(* CODESYS project SPT_MotionControl.library
   Placeholder: SPT Motion Control
   Title: SPT Motion Control
   Version: 3.1.0
   Company: Beckhoff Automation LLC

Project tree, tasks and I/O mapping:
  libraries: SPT Base Types, * (Beckhoff Automation LLC); Tc2_Math, * (Beckhoff Automation GmbH); Tc2_MC2, * (Beckhoff Automation GmbH); Tc2_MC2_Camming, * (Beckhoff Automation GmbH); Tc2_MC2_Drive, * (Beckhoff Automation GmbH); Tc2_Standard, * (Beckhoff Automation GmbH); Tc2_System, * (Beckhoff Automation GmbH); Tc3_MC2_AdvancedHoming, * (Beckhoff Automation GmbH); Tc3_Module, * (Beckhoff Automation GmbH)
  DUTs/
    data type E_CamAxisState
    data type E_CamSyncMode
    data type ST_AbsHomeParameters
    data type ST_CamParameters
    data type ST_CamPoints
    data type ST_StepBlockLagBasedParameters
  Function Blocks/
    Hardware Utilities/
      function block FB_ResetRoutine_CoEDrive [ST]: Axis, CyclicLogic, Execute
      function block FB_ResetRoutine_SoEDrive [ST]: Axis, CyclicLogic, Execute
    Homing Routines/
      function block FB_HomeRoutine_AbsHoming [ST]: Axis, CyclicLogic, Execute, Parameters
      function block FB_HomeRoutine_HardStop [ST]: Axis, CyclicLogic, Execute, HomePosition, Parameters
      function block FB_HomeRoutine_SetPosition [ST]: Axis, CyclicLogic, Execute, HomePosition
      function block FB_HomeRoutine_SetZeroHere [ST]: Axis, CyclicLogic, Execute
    function block FB_BasicAxis [ST]: Disable, Enable, Home, Jog, MoveAbsolute, MoveModulo, MoveRelative, MoveVelocity, Reset, Stop, WriteBoolParameter, WriteParameter, Acceleration, Deceleration, Jerk, Velocity, ActualAcceleration, ActualPosition, ActualPositionModulo, ActualTorque, ActualVelocity, PositionLag, SetAcceleration, SetPosition, SetPositionModulo, SetVelocity, Enabled, InPosition, Stopped, Axis, HomeMethod, InhibitFeedNegative, InhibitFeedPositive, Override, ResetMethod, CyclicLogic, CallFBs, Initialize, AxisParameters
    function block FB_BasicSlaveAxis [ST]: Home, MoveAbsolute, MoveModulo, MoveRelative, MoveVelocity, Reset, GearIn, GearOut, InGear, Master1, Master2, Master3, Master4, RatioMaster1, RatioMaster2, RatioMaster3, RatioMaster4, Stop, CyclicLogic, CallFBs, Initialize
    function block FB_CamSlaveAxis [ST]: Home, MoveModulo, Reset, Stop, CamParameters, ChangeMode, FindSlavePos, FindSyncPos, InSync, Master, RunningTable, StartCouple, StartSync, SyncPos, UpdateTable, CyclicLogic, CallFBs, Initialize
    function block FB_RingBuffer_MCMoveAbsolute [ST]: CurrentFB, GetNewFB
    function block FB_RingBuffer_MCMoveModulo [ST]: CurrentFB, GetNewFB
    function block FB_RingBuffer_MCMoveRelative [ST]: CurrentFB, GetNewFB
    function block FB_RingBuffer_MCMoveVelocity [ST]: CurrentFB, GetNewFB
  Interfaces/
    interface I_BasicAxis: Disable, Enable, Home, Jog, MoveAbsolute, MoveModulo, MoveRelative, MoveVelocity, Reset, Stop, WriteBoolParameter, WriteParameter, Acceleration, Deceleration, Jerk, Velocity, ActualAcceleration, ActualPosition, ActualPositionModulo, ActualTorque, ActualVelocity, PositionLag, SetAcceleration, SetPosition, SetPositionModulo, SetVelocity, Enabled, InPosition, Stopped, Axis, HomeMethod, InhibitFeedNegative, InhibitFeedPositive, Override, ResetMethod
    interface I_BasicSlaveAxis: GearIn, GearOut, InGear, Master1, Master2, Master3, Master4, RatioMaster1, RatioMaster2, RatioMaster3, RatioMaster4
    interface I_CamSlaveAxis: CamParameters, ChangeMode, FindSlavePos, FindSyncPos, InSync, Master, RunningTable, StartCouple, StartSync, SyncPos, UpdateTable
    interface I_MotionSequence: Axis, Execute
  Project Information/
    function F_GetCompany [ST]
    function F_GetTitle [ST]
    function F_GetVersion [ST]
  Version/
    global variables Global_Version
  global variables Parameters_MotionControl
*)

// DUTs/E_CamAxisState
{attribute 'qualified_only'}
{attribute 'strict'}
TYPE E_CamAxisState : (
        eCamAxisState_Disabled := 0,
        eCamAxisState_ReadMasterParameters,
        eCamAxisState_ReadSlaveParameters,
        eCamAxisState_AxisInitDone,
        eCamAxisState_WaitForCommand,
        eCamAxisState_DecoupleBeforeStart,
        eCamAxisState_CheckTableSelect,
        eCamAxisState_LoadCamTable,
        eCamAxisState_CheckAxisStatus,
        eCamAxisState_ReadSlaveDynamics,
        eCamAxisState_DetermineSyncMove,
        eCamAxisState_SlaveSyncMove,
        eCamAxisState_CoupleSlave,
        eCamAxisState_SetChangeMode,
        eCamAxisState_WaitForChangeCommand,
        eCamAxisState_WriteNewTable,
        eCamAxisState_WaitForActive,
        //eCamAxisState_DecoupleSlave,

        //eCamAxisState_HaltSlave,
        eCamAxisState_Error
    ) UDINT;
END_TYPE

// DUTs/E_CamSyncMode
{attribute 'qualified_only'}
{attribute 'strict'}
TYPE E_CamSyncMode : (
        eCamSyncMode_ShortestWay    := 0, // Move the Shortest Distance
        eCamSyncMode_Forward        := 1, // Move Only in the Forward Direction
        eCamSyncMode_Reverse        := 2, // Move Only in the Reverse Direction
        eCamSyncMode_Window_Forward := 3, // Move Shortest Distance If In Window Else Move Forward
        eCamSyncMode_Window_Reverse := 4  // Move Shortest Distance If In Window Else Move Reverse
    );
END_TYPE

// DUTs/ST_AbsHomeParameters
TYPE ST_AbsHomeParameters :
    STRUCT
        PositionBias           : LREAL;
        PositionLimit_Positive : LREAL;
        PositionLimit_Negative : LREAL;
    END_STRUCT
END_TYPE

// DUTs/ST_CamParameters
TYPE ST_CamParameters :
    STRUCT
        // Table Must Be Constructed of Motion Functions
        MasterPos    : LREAL         := 0.1;                                    // Position of Master For Which Corresponding Slave Position Is Found For
        SyncMode     : E_CamSyncMode := E_CamSyncMode.eCamSyncMode_ShortestWay; // Specifies Which Direction Slave Moves To Synchronize With the Master
        SyncWindow   : LREAL         := 10.0;                                   // Used In Conjunction With Sync Mode
        SyncVelocity : LREAL         := 10.0;                                   // Used When Slave Moves To Synchronization Position
        SyncAccel    : LREAL         := 100.0;                                  // Used When Slave Moves To Synchronization Position
        SyncDecel    : LREAL         := 100.0;                                  // Used When Slave Moves To Synchronization Position
        SyncJerk     : LREAL         := 1000.0;                                 // Used When Slave Moves To Synchronization Position

        //EmergencyDecel : LREAL         := 1000.0;                                 // Rate At Which Slave Stops On Loss of Function Block Enable or Error

        //EmergencyJerk  : LREAL         := 10000.0;                                // Rate At Which Slave Stops On Loss of Function Block Enable or Error
        TableSelect   : UDINT     := 1; // Selects Which of Five Cam Tables To Use
        CamTableId    : MC_CAM_ID := 1; // Make Sure All Your Id's are Unique
        CamTable      : ARRAY[1..Parameters_MotionControl.CAM_SLAVE_AXIS_TABLES] OF ST_CamPoints;
        Periodic      : BOOL         := TRUE;
        MasterOffset  : LREAL        := 0.0;
        SlaveOffset   : LREAL        := 0.0;
        MasterScaling : LREAL        := 1.0;
        SlaveScaling  : LREAL        := 1.0;
        StartMode     : MC_StartMode := MC_STARTMODE_ABSOLUTE;
        BufferMode    : MC_BufferMode;
        CamInOptions  : ST_CamInOptions;
        ChangeOptions : ST_CamInOptions; // Used for MC_SetCamOnlineChangeMode; Change Mode is Set After Cam In
    END_STRUCT
END_TYPE

// DUTs/ST_CamPoints
TYPE ST_CamPoints :
    STRUCT
        Points         : ARRAY[1..Parameters_MotionControl.CAM_SLAVE_AXIS_MAX_CAM_POINTS] OF MC_MotionFunctionPoint; // Array of Points 
        NumberOfPoints : DINT;                                                                                   // Quantity of Points 
    END_STRUCT
END_TYPE

// TYPE MC_MotionFunctionType

// 	MOTIONFUNCTYPE_NOTDEF,

//	MOTIONFUNCTYPE_POLYNOM1

//	MOTIONFUNCTYPE_POLYNOM3

//	MOTIONFUNCTYPE_POLYNOM5								Rest to Rest

//	MOTIONFUNCTYPE_POLYNOM8

// 	MOTIONFUNCTYPE_SINUSLINIE

//	MOTIONFUNCTYPE_MODSINUSLINIE

//	MOTIONFUNCTYPE_BESTEHORN

//	MOTIONFUNCTYPE_BESCHLTRAPEZ

//	MOTIONFUNCTYPE_POLYNOM5_MM						Motion to Motion

//	MOTIONFUNCTYPE_SINUS_GERADE_KOMBI

// 	MOTIONFUNCTYPE_HARMONIC_KOMBI_RT

//	MOTIONFUNCTYPE_HARMONIC_KOMBI_TR

//	MOTIONFUNCTYPE_HARMONIC_KOMBI_VT

//	MOTIONFUNCTYPE_HARMONIC_KOMBI_TV

//	MOTIONFUNCTYPE_BESCHLTRAPEZ_RT

//	MOTIONFUNCTYPE_BESCHLTRAPEZ_RT

//	MOTIONFUNCTYPE_MODSINUSLINIE_VV

//	MOTIONFUNCTYPE_POLYNOM7_MM

//	MOTIONFUNCTYPE_POLYNOM6STP

//	MOTIONFUNCTYPE_POLYNOM6WDP

//	MOTIONFUNCTYPE_STEPFUNCTION

// TYPE MC_MotionFunctionPoint

//	MOTIONPOINTTYPE_IGNORE

//	MOTIONPOINTTYPE_REST				Vel = 0 and Accel = 0

//	MOTIONPOINTTYPE_VELOCITY		Vel = V and Accel = 0

//	MOTIONPOINTTYPE_TURN				Vel = 0 and Accel = A

//	MOTIONPOINTTYPE_MOTION			Vel = V and Accel = A

//	MOTIONPOINTTYPE_ADD

//	MOTIONPOINTTYPE_ACTIVATION

// DUTs/ST_StepBlockLagBasedParameters
TYPE ST_StepBlockLagBasedParameters :
    STRUCT
        Direction              : MC_Home_Direction := mcNegativeDirection;
        Velocity               : LREAL             := 10;
        Acceleration           : LREAL             := 100;
        Deceleration           : LREAL             := 100;
        Jerk                   : LREAL             := 1000;
        DetectionVelocityLimit : LREAL             := 5;
        DetectionVelocityTime  : TIME              := T#500MS;
        TimeLimit              : TIME;
        DistanceLimit          : LREAL;
        TorqueLimit            : LREAL            := 10;
        LagLimit               : LREAL            := 10;
        Options                : ST_Home_Options3 := (InstantLagReduction := TRUE);
    END_STRUCT
END_TYPE

// Version/Global_Version
{attribute 'TcGenerated'}
{attribute 'no-analysis'}
{attribute 'linkalways'}
// This function has been automatically generated from the project information.
VAR_GLOBAL CONSTANT
	{attribute 'const_non_replaced'}
	stLibVersion_SPT_Motion_Control : ST_LibVersion := (iMajor := 3, iMinor := 1, iBuild := 0, iRevision := 0, nFlags := 1, sVersion := '3.1.0');
END_VAR

// Parameters_MotionControl
{attribute 'qualified_only'}
VAR_GLOBAL CONSTANT
    ALLOW_UNLINKED_NC_AXES : BOOL := FALSE;
	    CAM_SLAVE_AXIS_TABLES         : UDINT := 10;
    CAM_SLAVE_AXIS_MAX_CAM_POINTS : UDINT := 30;
END_VAR

// Function Blocks/Hardware Utilities/FB_ResetRoutine_CoEDrive
FUNCTION_BLOCK FINAL FB_ResetRoutine_CoEDrive EXTENDS FB_CyclicFB IMPLEMENTS I_MotionSequence
VAR_INPUT
END_VAR
VAR_OUTPUT
END_VAR
VAR
    _Axis : I_BasicAxis;
END_VAR

VAR
    MCReset : MC_Reset;
END_VAR

PROPERTY Axis : I_BasicAxis
GET
Axis := _Axis;
END_GET
SET
_Axis := Axis;
END_SET
END_PROPERTY

METHOD PUBLIC  CyclicLogic
VAR_INPUT
END_VAR
MCReset(Axis := _Axis.Axis, Busy => _Busy);

IF NOT MCReset.Busy THEN
    IF MCReset.Error THEN
        _Error   := TRUE;
        _ErrorID := MCReset.ErrorID;
    END_IF

    MCReset(Axis := _Axis.Axis, Execute := FALSE);
END_IF
END_METHOD

METHOD PUBLIC Execute : BOOL
IF (_Axis = 0) THEN
    RETURN;
END_IF

MCReset(Axis := _Axis.Axis, Execute := TRUE);

_Busy    := TRUE;
_Error   := FALSE;
_ErrorID := 0;

Execute := TRUE;
END_METHOD

END_FUNCTION_BLOCK

// Interfaces/I_MotionSequence
INTERFACE I_MotionSequence EXTENDS I_CyclicFB

PROPERTY Axis : I_BasicAxis
GET
END_GET
SET
END_SET
END_PROPERTY

METHOD Execute : BOOL
END_METHOD

END_INTERFACE

// Interfaces/I_BasicAxis
INTERFACE I_BasicAxis EXTENDS I_CyclicFB

METHOD PUBLIC Disable : BOOL
VAR_INPUT
END_VAR
END_METHOD

METHOD PUBLIC Enable : BOOL
VAR_INPUT
END_VAR
END_METHOD

METHOD PUBLIC Home : BOOL
VAR_INPUT
END_VAR
END_METHOD

METHOD Jog : BOOL
VAR_INPUT
    JogFW    : BOOL;
    JogBW    : BOOL;
    JogMode  : E_JogMode;
    Position : LREAL;
END_VAR
END_METHOD

METHOD PUBLIC MoveAbsolute : BOOL
VAR_INPUT
    Position      : LREAL;
    AbortPrevious : BOOL;
END_VAR
END_METHOD

METHOD MoveModulo : BOOL
VAR_INPUT
    Position      : LREAL;
    Direction     : MC_Direction;
    AbortPrevious : BOOL;
END_VAR
END_METHOD

METHOD PUBLIC MoveRelative : BOOL
VAR_INPUT
    Distance      : LREAL;
    AbortPrevious : BOOL;
END_VAR
END_METHOD

METHOD MoveVelocity : BOOL
VAR_INPUT
    Velocity      : LREAL;
    AbortPrevious : BOOL;
END_VAR
END_METHOD

METHOD PUBLIC Reset : BOOL
END_METHOD

METHOD Stop : BOOL
END_METHOD

METHOD WriteBoolParameter : BOOL
VAR_INPUT
    ParameterNumber : MC_AxisParameter;
    Value           : BOOL;
END_VAR
END_METHOD

METHOD WriteParameter : BOOL
VAR_INPUT
    ParameterNumber : MC_AxisParameter;
    Value           : LREAL;
END_VAR
END_METHOD

PROPERTY Acceleration : LREAL
GET
END_GET
SET
END_SET
END_PROPERTY

PROPERTY Deceleration : LREAL
GET
END_GET
SET
END_SET
END_PROPERTY

PROPERTY Jerk : LREAL
GET
END_GET
SET
END_SET
END_PROPERTY

PROPERTY Velocity : LREAL
GET
END_GET
SET
END_SET
END_PROPERTY

PROPERTY ActualAcceleration : LREAL
GET
END_GET
END_PROPERTY

PROPERTY ActualPosition : LREAL
GET
END_GET
END_PROPERTY

PROPERTY ActualPositionModulo : LREAL
GET
END_GET
END_PROPERTY

PROPERTY ActualTorque : LREAL
GET
END_GET
END_PROPERTY

PROPERTY ActualVelocity : LREAL
GET
END_GET
END_PROPERTY

PROPERTY PositionLag : LREAL
GET
END_GET
END_PROPERTY

PROPERTY SetAcceleration : LREAL
GET
END_GET
END_PROPERTY

PROPERTY SetPosition : LREAL
GET
END_GET
END_PROPERTY

PROPERTY SetPositionModulo : LREAL
GET
END_GET
END_PROPERTY

PROPERTY SetVelocity : LREAL
GET
END_GET
END_PROPERTY

PROPERTY Enabled : BOOL
GET
END_GET
END_PROPERTY

PROPERTY InPosition : BOOL
GET
END_GET
END_PROPERTY

PROPERTY Stopped : BOOL
GET
END_GET
END_PROPERTY

PROPERTY Axis : REFERENCE TO AXIS_REF
GET
END_GET
END_PROPERTY

PROPERTY HomeMethod : I_MotionSequence
SET
END_SET
END_PROPERTY

PROPERTY InhibitFeedNegative : BOOL
SET
END_SET
END_PROPERTY

PROPERTY InhibitFeedPositive : BOOL
SET
END_SET
END_PROPERTY

PROPERTY Override : LREAL
GET
END_GET
SET
END_SET
END_PROPERTY

PROPERTY ResetMethod : I_MotionSequence
SET
END_SET
END_PROPERTY

END_INTERFACE

// Function Blocks/Hardware Utilities/FB_ResetRoutine_SoEDrive
FUNCTION_BLOCK FINAL FB_ResetRoutine_SoEDrive EXTENDS FB_CyclicFB IMPLEMENTS I_MotionSequence
VAR_INPUT
END_VAR
VAR_OUTPUT
END_VAR
VAR
    _Axis : I_BasicAxis;
END_VAR

VAR
    MCReset      : MC_Reset;
    SoEReset     : FB_SoEReset;
    SequenceStep : UDINT;
END_VAR

PROPERTY Axis : I_BasicAxis
GET
Axis := _Axis;
END_GET
SET
_Axis := Axis;
END_SET
END_PROPERTY

METHOD PUBLIC  CyclicLogic
VAR_INPUT
END_VAR
CASE SequenceStep OF
    10:
        SoEReset(Axis := _Axis.Axis, Execute := TRUE);

        IF NOT SoEReset.Busy THEN
            IF SoEReset.Error THEN
                _Error := TRUE;

                IF SoEReset.SercosErrId < 0 THEN
                    _ErrorID := SoEReset.SercosErrId;
                ELSE
                    _ErrorID := SoEReset.AdsErrId;
                END_IF

                SequenceStep := 0;
            ELSE
                //No error occurred
                SequenceStep := SequenceStep + 10;
            END_IF

            SoEReset(Axis := _Axis.Axis, Execute := FALSE);
        END_IF

    20:
        MCReset(Axis := _Axis.Axis, Execute := TRUE);

        IF NOT MCReset.Busy THEN
            IF MCReset.Error THEN
                _Error   := TRUE;
                _ErrorID := MCReset.ErrorID;
            END_IF

            //Done
            SequenceStep := 0;
            MCReset(Axis := _Axis.Axis, Execute := FALSE);
        END_IF
END_CASE

_Busy := SequenceStep <> 0;
END_METHOD

METHOD PUBLIC Execute : BOOL
IF (_Axis = 0) OR _Busy THEN
    RETURN;
END_IF

_Busy        := TRUE;
_Error       := FALSE;
_ErrorID     := 0;
SequenceStep := 10;

Execute := TRUE;
END_METHOD

END_FUNCTION_BLOCK

// Function Blocks/Homing Routines/FB_HomeRoutine_AbsHoming
FUNCTION_BLOCK FB_HomeRoutine_AbsHoming EXTENDS FB_CyclicFB IMPLEMENTS I_MotionSequence
VAR
    _Axis : I_BasicAxis;
END_VAR

VAR
    _HomingDn                 : BOOL;
    _Reset                    : BOOL;
    _Parameters               : REFERENCE TO ST_AbsHomeParameters;
    SequenceStep              : UDINT;
    ReadWatchdog              : TON;
    WriteWatchdog             : TON;
    McReadParameter_Bias      : MC_ReadParameter;
    McWriteParameter_Bias     : MC_WriteParameter;
    McWriteParameter_SwPosLim : MC_WriteParameter;
    McWriteParameter_SwNegLim : MC_WriteParameter;
    McHome                    : MC_Home;
    CurrentPositionBias       : LREAL;
END_VAR

//There should be no code in the function block body

PROPERTY Axis : I_BasicAxis
GET
Axis := _Axis;
END_GET
SET
_Axis := Axis;
END_SET
END_PROPERTY

METHOD CyclicLogic
VAR_INPUT
END_VAR
IF __ISVALIDREF(_Parameters) THEN
    CASE SequenceStep OF
        0: (* Init State *)
            _Busy                             := TRUE;
            ReadWatchdog.IN                   := FALSE;
            WriteWatchdog.IN                  := TRUE;
            McReadParameter_Bias.Enable       := FALSE;
            McWriteParameter_Bias.Execute     := TRUE;
            McWriteParameter_SwPosLim.Execute := TRUE;
            McWriteParameter_SwNegLim.Execute := TRUE;
            SequenceStep                      := 10;
        10: (* Wait for init done *)

            // check for errors
            IF WriteWatchdog.Q THEN
                SequenceStep := 500;
                _Error       := TRUE;
                _ErrorID     := 10;
            ELSIF McWriteParameter_Bias.Error THEN
                SequenceStep := 500;
                _Error       := TRUE;
                _ErrorID     := McWriteParameter_Bias.ErrorID;
            ELSIF McWriteParameter_SwPosLim.Error THEN
                SequenceStep := 500;
                _Error       := TRUE;
                _ErrorID     := McWriteParameter_SwPosLim.ErrorID;
            ELSIF McWriteParameter_SwNegLim.Error THEN
                SequenceStep := 500;
                _Error       := TRUE;
                _ErrorID     := McWriteParameter_SwNegLim.ErrorID;
            END_IF

            IF (McWriteParameter_Bias.Done AND McWriteParameter_SwPosLim.Done AND McWriteParameter_SwNegLim.Done) THEN
                WriteWatchdog.IN := FALSE;
                McHome.Execute   := TRUE;
                _Busy            := FALSE;
            END_IF
        20: (* Reads the Position Bias Variable *)
            _Busy                             := TRUE;
            WriteWatchdog.IN                  := FALSE;
            McWriteParameter_Bias.Execute     := FALSE;
            McWriteParameter_SwPosLim.Execute := FALSE;
            McWriteParameter_SwNegLim.Execute := FALSE;

            (* 1042 = Axis Encoder Offset ... AKA: Position Bias *)
            IF NOT McReadParameter_Bias.Enable THEN
                ReadWatchdog.IN             := TRUE;
                McReadParameter_Bias.Enable := TRUE;
            END_IF

            IF (McReadParameter_Bias.Enable AND McReadParameter_Bias.Valid) THEN
                ReadWatchdog.IN             := FALSE;
                McReadParameter_Bias.Enable := FALSE;

                (* Do the calculations to figure how far to adjust the Position Bias # *)

                (* Write Value back to the bias for the new teach position *)
                _Parameters.PositionBias := CurrentPositionBias + (_Axis.Axis.NcToPlc.ActPos * -1.0);
                SequenceStep             := 30;
            ELSIF McReadParameter_Bias.Error THEN
                SequenceStep := 500;
                _Error       := TRUE;
                _ErrorID     := McReadParameter_Bias.ErrorID;
            ELSIF ReadWatchdog.Q THEN
                SequenceStep := 500;
                _Error       := TRUE;
                _ErrorID     := 20;
            END_IF
        30:
            _Busy                             := TRUE;
            WriteWatchdog.IN                  := TRUE;
            McWriteParameter_Bias.Execute     := TRUE;
            McWriteParameter_SwPosLim.Execute := TRUE;
            McWriteParameter_SwNegLim.Execute := TRUE;
            SequenceStep                      := 10;
        500: (* Error State *)
            _Busy                             := FALSE;
            ReadWatchdog.IN                   := FALSE;
            WriteWatchdog.IN                  := FALSE;
            McReadParameter_Bias.Enable       := FALSE;
            McWriteParameter_Bias.Execute     := FALSE;
            McWriteParameter_SwPosLim.Execute := FALSE;
            McWriteParameter_SwNegLim.Execute := FALSE;
    END_CASE
ELSE
    _Busy                             := FALSE;
    _Error                            := FALSE;
    _ErrorID                          := 0;
    SequenceStep                      := 0;
    ReadWatchdog.IN                   := FALSE;
    WriteWatchdog.IN                  := FALSE;
    McReadParameter_Bias.Enable       := FALSE;
    McWriteParameter_Bias.Execute     := FALSE;
    McWriteParameter_SwPosLim.Execute := FALSE;
    McWriteParameter_SwNegLim.Execute := FALSE;
END_IF

ReadWatchdog(PT := T#1S);
WriteWatchdog(PT := T#1S);
McHome(Axis := _Axis.Axis, HomingMode := MC_ForceCalibration);

(* Position Bias Reading *)
McReadParameter_Bias(ParameterNumber := MC_AxisParameter.AxisEncoderOffset, (*AxisEncoderOffset*)
                     Axis            := _Axis.Axis,
                     Value           => CurrentPositionBias);

(* Writes the Position Bias Variable *)
McWriteParameter_Bias(Execute         := McWriteParameter_Bias.Execute,
                      ParameterNumber := MC_AxisParameter.AxisEncoderOffset, (*AxisEncoderOffset*)
                      Value           := _Parameters.PositionBias,
                      Axis            := _Axis.Axis);

(* Writes the SW Positive Limit Variable *)
McWriteParameter_SwPosLim(Execute         := McWriteParameter_SwPosLim.Execute,
                          ParameterNumber := MC_AxisParameter.SWLimitPos,
                          Value           := _Parameters.PositionLimit_Positive,
                          Axis            := _Axis.Axis);

(* Writes the SW Negetive Limit Variable *)
McWriteParameter_SwNegLim(Execute         := McWriteParameter_SwNegLim.Execute,
                          ParameterNumber := MC_AxisParameter.SWLimitNeg,
                          Value           := _Parameters.PositionLimit_Negative,
                          Axis            := _Axis.Axis);
END_METHOD

METHOD Execute : BOOL
IF (_Axis = 0) OR _Busy OR NOT (McWriteParameter_Bias.Done AND McWriteParameter_SwPosLim.Done AND McWriteParameter_SwNegLim.Done) THEN
    RETURN;
END_IF

_Busy        := TRUE;
_Error       := FALSE;
_ErrorID     := 0;
_HomingDn    := FALSE;
SequenceStep := 20;
Execute      := TRUE;
END_METHOD

PROPERTY Parameters : REFERENCE TO ST_AbsHomeParameters
GET
IF __ISVALIDREF(_Parameters) THEN
    Parameters REF= _Parameters;
END_IF
END_GET
SET
_Parameters ref= Parameters;
END_SET
END_PROPERTY

END_FUNCTION_BLOCK

// Function Blocks/Homing Routines/FB_HomeRoutine_HardStop
FUNCTION_BLOCK FINAL FB_HomeRoutine_HardStop EXTENDS FB_CyclicFB IMPLEMENTS I_MotionSequence
VAR
    _Axis : I_BasicAxis;
END_VAR

VAR
    MCStepBlock    : MC_StepBlockLagBasedDetection;
    MCHomeDirect   : MC_HomeDirect;
    MCReset        : MC_Reset;
    MCAbortHoming  : MC_AbortHoming;
    AxisParameters : MC_HomingParameter;
    _Parameters    : ST_StepBlockLagBasedParameters;
    _HomePosition  : LREAL;
    SequenceStep   : UDINT;
END_VAR

//There should be no code in the function block body

PROPERTY Axis : I_BasicAxis
GET
Axis := _Axis;
END_GET
SET
_Axis := Axis;
END_SET
END_PROPERTY

METHOD PUBLIC CyclicLogic
CASE SequenceStep OF
    10:
        MCStepBlock(Axis                   := _Axis.Axis,
                    Parameter              := AxisParameters,
                    Execute                := TRUE,
                    Direction              := _Parameters.Direction,
                    Velocity               := _Parameters.Velocity,
                    Acceleration           := _Parameters.Acceleration,
                    Deceleration           := _Parameters.Deceleration,
                    Jerk                   := _Parameters.Jerk,
                    DetectionVelocityLimit := _Parameters.DetectionVelocityLimit,
                    DetectionVelocityTime  := _Parameters.DetectionVelocityTime,
                    TimeLimit              := _Parameters.TimeLimit,
                    DistanceLimit          := _Parameters.DistanceLimit,
                    TorqueLimit            := _Parameters.TorqueLimit,
                    LagLimit               := _Parameters.LagLimit,
                    Options                := _Parameters.Options);

        IF NOT MCStepBlock.Busy THEN
            IF MCStepBlock.Error THEN
                _Error       := TRUE;
                _ErrorID     := MCStepBlock.ErrorID;
                SequenceStep := 999;
            ELSE
                //No error occurred
                SequenceStep := SequenceStep + 10;
            END_IF

            MCStepBlock(Axis := _Axis.Axis, Parameter := AxisParameters, Execute := FALSE);
        END_IF
    20:
        MCHomeDirect(Axis        := _Axis.Axis,
                     Parameter   := AxisParameters,
                     Execute     := TRUE,
                     SetPosition := _HomePosition);

        IF NOT MCHomeDirect.Busy THEN
            IF MCHomeDirect.Error THEN
                _Error       := TRUE;
                _ErrorID     := MCHomeDirect.ErrorID;
                SequenceStep := 999;
            END_IF

            //Done
            SequenceStep := 0;
            MCHomeDirect(Axis := _Axis.Axis, Parameter := AxisParameters, Execute := FALSE);
        END_IF
    999:
        //An error occurred above--clear out position lag so we don't fault the axis with AbortHoming
        MCReset(Axis := _Axis.Axis, Execute := TRUE);
        IF NOT MCReset.Busy THEN
            //If this errors there's not much we can do about it
            SequenceStep := 1000;
            MCReset(Axis := _Axis.Axis, Execute := FALSE);
        END_IF
    1000:
        MCAbortHoming(Axis := _Axis.Axis, Parameter := AxisParameters, Execute := TRUE);
        IF NOT MCAbortHoming.Busy THEN
            IF MCAbortHoming.Error THEN
                _Error       := TRUE;
                _ErrorID     := MCAbortHoming.ErrorID;
                SequenceStep := 0;
            ELSE
                //No error occurred
                SequenceStep := 0;
            END_IF

            MCAbortHoming(Axis := _Axis.Axis, Parameter := AxisParameters, Execute := FALSE);
        END_IF
END_CASE

_Busy := SequenceStep <> 0;
END_METHOD

METHOD PUBLIC Execute : BOOL
IF (_Axis = 0) OR _Busy THEN
    RETURN;
END_IF

_Busy        := TRUE;
_Error       := FALSE;
_ErrorID     := 0;
SequenceStep := 10;
Execute      := TRUE;
END_METHOD

PROPERTY HomePosition : LREAL
GET
HomePosition := _HomePosition;
END_GET
SET
_HomePosition := HomePosition;
END_SET
END_PROPERTY

PROPERTY Parameters : ST_StepBlockLagBasedParameters
GET
Parameters := _Parameters;
END_GET
SET
_Parameters := Parameters;
END_SET
END_PROPERTY

END_FUNCTION_BLOCK

// Function Blocks/Homing Routines/FB_HomeRoutine_SetPosition
FUNCTION_BLOCK FINAL FB_HomeRoutine_SetPosition EXTENDS FB_CyclicFB IMPLEMENTS I_MotionSequence
VAR_INPUT
END_VAR

VAR_OUTPUT
END_VAR

VAR
    _Axis : I_BasicAxis;
END_VAR

VAR
    MCSetPosition : MC_SetPosition;
END_VAR

//There should be no code in the function block body

PROPERTY Axis : I_BasicAxis
GET
Axis := _Axis;
END_GET
SET
_Axis := Axis;
END_SET
END_PROPERTY

METHOD PUBLIC CyclicLogic
MCSetPosition(Axis := _Axis.Axis, Busy => _Busy);
IF NOT MCSetPosition.Busy THEN
    IF MCSetPosition.Error THEN
        _Error   := TRUE;
        _ErrorID := MCSetPosition.ErrorID;
    END_IF

    MCSetPosition(Axis := _Axis.Axis, Execute := FALSE);
END_IF
END_METHOD

METHOD PUBLIC Execute : BOOL
IF (_Axis = 0) THEN
    RETURN;
END_IF

MCSetPosition(Axis := _Axis.Axis, Execute := TRUE, Mode := FALSE);
_Error   := FALSE;
_ErrorID := 0;
Execute  := TRUE;
END_METHOD

PROPERTY HomePosition : LREAL
GET
HomePosition := MCSetPosition.Position;
END_GET
SET
MCSetPosition.Position := HomePosition;
END_SET
END_PROPERTY

END_FUNCTION_BLOCK

// Function Blocks/Homing Routines/FB_HomeRoutine_SetZeroHere
FUNCTION_BLOCK FINAL FB_HomeRoutine_SetZeroHere EXTENDS FB_CyclicFB IMPLEMENTS I_MotionSequence
VAR_INPUT
END_VAR

VAR_OUTPUT
END_VAR

VAR
    _Axis : I_BasicAxis;
END_VAR

VAR
    MCSetPosition : MC_SetPosition;
END_VAR

//There should be no code in the function block body

PROPERTY Axis : I_BasicAxis
GET
Axis := _Axis;
END_GET
SET
_Axis := Axis;
END_SET
END_PROPERTY

METHOD PUBLIC CyclicLogic
MCSetPosition(Axis := _Axis.Axis, Busy => _Busy);
IF NOT MCSetPosition.Busy THEN
    IF MCSetPosition.Error THEN
        _Error   := TRUE;
        _ErrorID := MCSetPosition.ErrorID;
    END_IF

    MCSetPosition(Axis := _Axis.Axis, Execute := FALSE);
END_IF
END_METHOD

METHOD PUBLIC Execute : BOOL
IF (_Axis = 0) THEN
    RETURN;
END_IF

MCSetPosition(Axis     := _Axis.Axis,
              Execute  := TRUE,
              Position := 0.0,
              Mode     := FALSE);

_Error   := FALSE;
_ErrorID := 0;
Execute  := TRUE;
END_METHOD

END_FUNCTION_BLOCK

// Function Blocks/FB_BasicAxis
FUNCTION_BLOCK FB_BasicAxis EXTENDS FB_CyclicFB IMPLEMENTS I_BasicAxis
VAR
    _Axis           		: AXIS_REF;
    _Velocity       		: LREAL;
    _Acceleration  			: LREAL;
    _Deceleration   		: LREAL;
    _Jerk          	 		: LREAL;
    ipHomeMethod    		: I_MotionSequence;
    ipResetMethod   		: I_MotionSequence;
    _AxisParameters 		: ST_AxisParameterSet;
	_InhibitFeedNegative	: BOOL := FALSE;
	_InhibitFeedPositive	: BOOL := FALSE;
	_ActualSuperPosVeloDiff	: LREAL;
	_ActualSuperPosDistance	: LREAL;
	_ActualSuperPosLength	: LREAL;
	_ActualSuperPosAccel	: LREAL;
	_ActualSuperPosDecel	: LREAL;
	_SuperPosBusy			: BOOL;
	_SuperPosDone			: BOOL;
	_SuperPosAborted		: BOOL;
    _Warning   				: BOOL;
    _WarningID 				: UDINT;
END_VAR

VAR
    MCPower                   : MC_Power;
    RingBuffer_MCMoveAbsolute : FB_RingBuffer_MCMoveAbsolute;
    RingBuffer_MCMoveRelative : FB_RingBuffer_MCMoveRelative;
    RingBuffer_MCMoveVelocity : FB_RingBuffer_MCMoveVelocity;
    RingBuffer_MCMoveModulo   : FB_RingBuffer_MCMoveModulo;
    MCMoveAbsolute            : POINTER TO MC_MoveAbsolute;
    MCMoveRelative            : POINTER TO MC_MoveRelative;
    MCMoveVelocity            : POINTER TO MC_MoveVelocity;
    MCMoveModulo              : POINTER TO MC_MoveModulo;
    //MCMoveSuperimposed		  : MC_MoveSuperimposed;
	//MCAbortSuperposition	  : MC_AbortSuperposition;
    MCJog                     : MC_Jog;
    MCHalt                    : MC_Halt;
    DefaultHome               : FB_HomeRoutine_SetZeroHere;
    DefaultReset              : FB_ResetRoutine_CoEDrive;
    MCReadParameterSet        : MC_ReadParameterSet;
    MCWriteParameter          : MC_WriteParameterPersistent;
    MCWriteBoolParameter      : MC_WriteBoolParameterPersistent;
    HomePreviouslyErrored     : BOOL;
    ResetPreviouslyErrored    : BOOL;
END_VAR

//There should be no code in the function block body

METHOD Disable : BOOL
MCPower(Axis            := _Axis,
        Enable          := FALSE);

Disable := TRUE;
END_METHOD

METHOD Enable : BOOL
IF _Error THEN
    RETURN;
END_IF

MCPower(Axis            := _Axis,
        Enable          := TRUE);
Enable := TRUE;
END_METHOD

METHOD Home : BOOL
IF _Busy OR _Error OR ipHomeMethod = 0 THEN
    RETURN;
END_IF

//This is used to trap circular errors (I_MotionStratery resets error bit on next execute)
HomePreviouslyErrored := FALSE;
ipHomeMethod.Execute();
Home := TRUE;
END_METHOD

METHOD Jog : BOOL
VAR_INPUT
    JogFW    : BOOL;
    JogBW    : BOOL;
    JogMode  : E_JogMode;
    Position : LREAL;
END_VAR
IF _Error THEN
    RETURN;
END_IF

MCJog(Axis         := _Axis,
      JogForward   := JogFW,
      JogBackwards := JogBW,
      Mode         := JogMode,
      Position     := Position,
      Velocity     := _Velocity,
      Acceleration := _Acceleration,
      Deceleration := _Deceleration,
      Jerk         := _Jerk);
END_METHOD

METHOD MoveAbsolute : BOOL
VAR_INPUT
    Position      : LREAL;
    AbortPrevious : BOOL;
END_VAR
IF _Error THEN
    RETURN;
ELSE
    IF (_Busy AND NOT AbortPrevious) THEN
        RETURN;
    END_IF
END_IF

MCMoveAbsolute := RingBuffer_MCMoveAbsolute.GetNewFB();
MCMoveAbsolute^(Axis         := _Axis,
                Execute      := TRUE,
                Position     := Position,
                Velocity     := _Velocity,
                Acceleration := _Acceleration,
                Deceleration := _Deceleration,
                Jerk         := _Jerk);

MoveAbsolute := TRUE;
END_METHOD

METHOD MoveModulo : BOOL
VAR_INPUT
    Position      : LREAL;
    Direction     : MC_Direction;
    AbortPrevious : BOOL;
END_VAR
IF _Error THEN
    RETURN;
ELSE
    IF (_Busy AND NOT AbortPrevious) THEN
        RETURN;
    END_IF
END_IF

MCMoveModulo := RingBuffer_MCMoveModulo.GetNewFB();
MCMoveModulo^(Axis         := _Axis,
              Execute      := TRUE,
              Position     := Position,
              Velocity     := _Velocity,
              Acceleration := _Acceleration,
              Deceleration := _Deceleration,
              Jerk         := _Jerk,
              Direction    := Direction);

MoveModulo := TRUE;
END_METHOD

METHOD MoveRelative : BOOL
VAR_INPUT
    Distance      : LREAL;
    AbortPrevious : BOOL;
END_VAR
IF _Error THEN
    RETURN;
ELSE
    IF (_Busy AND NOT AbortPrevious) THEN
        RETURN;
    END_IF
END_IF

MCMoveRelative := RingBuffer_MCMoveRelative.GetNewFB();
MCMoveRelative^(Axis         := _Axis,
                Execute      := TRUE,
                Distance     := Distance,
                Velocity     := _Velocity,
                Acceleration := _Acceleration,
                Deceleration := _Deceleration,
                Jerk         := _Jerk);

MoveRelative := TRUE;
END_METHOD

METHOD MoveVelocity : BOOL
VAR_INPUT
    Velocity      : LREAL;
    AbortPrevious : BOOL;
END_VAR
IF _Error THEN
    RETURN;
ELSE
    IF (_Busy AND NOT AbortPrevious) THEN
        RETURN;
    END_IF
END_IF

IF ABS(Velocity) > _AxisParameters.fVeloMaximum THEN
    Trace('Velocity setpoint exceeds axis limit');
END_IF

IF Velocity < 0 THEN
    MCMoveVelocity            := RingBuffer_MCMoveVelocity.GetNewFB();
    MCMoveVelocity^.Direction := MC_Negative_Direction;
ELSE
    MCMoveVelocity            := RingBuffer_MCMoveVelocity.GetNewFB();
    MCMoveVelocity^.Direction := MC_Positive_Direction;
END_IF

_Velocity := ABS(Velocity);
MCMoveVelocity^(Axis         := _Axis,
                Execute      := TRUE,
                Velocity     := Velocity,
                Acceleration := _Acceleration,
                Deceleration := _Deceleration,
                Jerk         := _Jerk);

MoveVelocity := TRUE;
END_METHOD

METHOD Reset : BOOL
IF _Busy OR ipResetMethod = 0 THEN
    RETURN;
END_IF

//This is used to trap circular errors (I_MotionStratery resets error bit on next execute)
ResetPreviouslyErrored := FALSE;
IF ipResetMethod.Execute() THEN
    IF MCMoveAbsolute <> 0 THEN
        IF MCMoveAbsolute^.Error THEN
            MCMoveAbsolute^(Axis := _Axis, Execute := FALSE);
        END_IF
    END_IF

    IF MCMoveRelative <> 0 THEN
        IF MCMoveRelative^.Error THEN
            MCMoveRelative^(Axis := _Axis, Execute := FALSE);
        END_IF
    END_IF

    IF MCMoveVelocity <> 0 THEN
        IF MCMoveVelocity^.Error THEN
            MCMoveVelocity^(Axis := _Axis, Execute := FALSE);
        END_IF
    END_IF

    IF MCMoveModulo <> 0 THEN
        IF MCMoveModulo^.Error THEN
            MCMoveModulo^(Axis := _Axis, Execute := FALSE);
        END_IF
    END_IF

    IF MCHalt.Error THEN
        MCHalt(Axis := _Axis, Execute := FALSE);
    END_IF
	
//    IF MCMoveSuperimposed.Error THEN
//        MCMoveSuperimposed(Axis := _Axis, Execute := FALSE);
//    END_IF
	
//    IF MCAbortSuperposition.Error THEN
//        MCAbortSuperposition(Axis := _Axis, Execute := FALSE);
//    END_IF  

    IF MCReadParameterSet.Error THEN
        MCReadParameterSet(Axis := _Axis, Parameter := _AxisParameters, Execute := FALSE);
    END_IF

    IF MCWriteBoolParameter.Error THEN
        MCWriteBoolParameter(Axis := _Axis, Execute := FALSE);
    END_IF

    IF MCWriteParameter.Error THEN
        MCWriteParameter(Axis := _Axis, Execute := FALSE);
    END_IF

    _Error   	:= FALSE;
    _ErrorID 	:= 0;
    _Warning   	:= FALSE;
    _WarningID 	:= 0;
    Reset    	:= TRUE;
END_IF
END_METHOD

METHOD Stop : BOOL
IF _Error AND _Axis.Status.Error THEN
    (* It's possible that a function block errored but
	not the NC itself--in this case we can allow a stop command.
	If the NC axis has a real fault then we want a successful reset first *)
    RETURN;
END_IF

MCHalt(Axis         := _Axis,
       Execute      := TRUE,
       Deceleration := _Deceleration,
       Jerk         := _Jerk);

Stop := TRUE;
END_METHOD

METHOD WriteBoolParameter : BOOL
VAR_INPUT
    ParameterNumber : MC_AxisParameter;
    Value           : BOOL;
END_VAR
IF _Busy OR _Error THEN
    RETURN;
END_IF

MCWriteBoolParameter(Axis            := _Axis,
                     Execute         := TRUE,
                     ParameterNumber := ParameterNumber,
                     Value           := Value);

WriteBoolParameter := TRUE;
END_METHOD

METHOD WriteParameter : BOOL
VAR_INPUT
    ParameterNumber : MC_AxisParameter;
    Value           : LREAL;
END_VAR
IF _Busy OR _Error THEN
    RETURN;
END_IF

MCWriteParameter(Axis            := _Axis,
                 Execute         := TRUE,
                 ParameterNumber := ParameterNumber,
                 Value           := Value);

WriteParameter := TRUE;
END_METHOD

PROPERTY Acceleration : LREAL
GET
Acceleration := _Acceleration;
END_GET
SET
IF Acceleration > _AxisParameters.fAccelerationMax THEN
    Trace('Acceleration setpoint exceeds axis limit');
END_IF

_Acceleration := Acceleration;
END_SET
END_PROPERTY

PROPERTY Deceleration : LREAL
GET
Deceleration := _Deceleration;
END_GET
SET
IF Deceleration > _AxisParameters.fDecelerationMax THEN
    Trace('Deceleration setpoint exceeds axis limit');
END_IF

_Deceleration := Deceleration;
END_SET
END_PROPERTY

PROPERTY Jerk : LREAL
GET
Jerk := _Jerk;
END_GET
SET
_Jerk := Jerk;
END_SET
END_PROPERTY

PROPERTY Velocity : LREAL
GET
Velocity := _Velocity;
END_GET
SET
IF Velocity > _AxisParameters.fVeloMaximum THEN
    Trace('Velocity setpoint exceeds axis limit');
END_IF

_Velocity := Velocity;
END_SET
END_PROPERTY

PROPERTY ActualAcceleration : LREAL
GET
ActualAcceleration := Axis.NcToPlc.ActAcc;
END_GET
END_PROPERTY

PROPERTY ActualPosition : LREAL
GET
ActualPosition := Axis.NcToPlc.ActPos;
END_GET
END_PROPERTY

PROPERTY ActualPositionModulo : LREAL
GET
ActualPositionModulo := Axis.NcToPlc.ModuloActPos;
END_GET
END_PROPERTY

PROPERTY ActualTorque : LREAL
GET
ActualTorque := Axis.NcToPlc.ActTorque;
END_GET
END_PROPERTY

PROPERTY ActualVelocity : LREAL
GET
ActualVelocity := Axis.NcToPlc.ActVelo;
END_GET
END_PROPERTY

PROPERTY PositionLag : LREAL
GET
PositionLag := Axis.NcToPlc.PosDiff;
END_GET
END_PROPERTY

PROPERTY SetAcceleration : LREAL
GET
SetAcceleration := Axis.NcToPlc.SetAcc;
END_GET
END_PROPERTY

PROPERTY SetPosition : LREAL
GET
SetPosition := Axis.NcToPlc.SetPos;
END_GET
END_PROPERTY

PROPERTY SetPositionModulo : LREAL
GET
SetPositionModulo := Axis.NcToPlc.ModuloSetPos;
END_GET
END_PROPERTY

PROPERTY SetVelocity : LREAL
GET
SetVelocity := Axis.NcToPlc.SetVelo;
END_GET
END_PROPERTY

PROPERTY Enabled : BOOL
GET
Enabled := MCPower.Status;
END_GET
END_PROPERTY

PROPERTY InPosition : BOOL
GET
InPosition := _Axis.Status.InTargetPosition;
END_GET
END_PROPERTY

PROPERTY Stopped : BOOL
GET
Stopped := _Axis.Status.NotMoving OR _Axis.Status.Disabled;
END_GET
END_PROPERTY

PROPERTY Axis : REFERENCE TO AXIS_REF
GET
Axis REF= _Axis;
END_GET
END_PROPERTY

PROPERTY HomeMethod : I_MotionSequence
GET
HomeMethod := ipHomeMethod;
END_GET
SET
ipHomeMethod      := HomeMethod;
ipHomeMethod.Axis := THIS^;
END_SET
END_PROPERTY

PROPERTY InhibitFeedNegative : BOOL
SET
_InhibitFeedNegative := InhibitFeedNegative;
END_SET
END_PROPERTY

PROPERTY InhibitFeedPositive : BOOL
SET
_InhibitFeedPositive := InhibitFeedPositive;
END_SET
END_PROPERTY

PROPERTY Override : LREAL
GET
Override := MCPower.Override;
END_GET
SET
IF Override >= 0 AND Override <= 100 THEN
    MCPower.Override := Override;
END_IF
END_SET
END_PROPERTY

PROPERTY ResetMethod : I_MotionSequence
GET
ResetMethod := ipResetMethod;
END_GET
SET
ipResetMethod      := ResetMethod;
ipResetMethod.Axis := THIS^;
END_SET
END_PROPERTY

METHOD PUBLIC CyclicLogic
VAR_INPUT
END_VAR
IF NOT _InitComplete THEN
    _InitComplete := THIS^.Initialize();
    RETURN;
END_IF

//Call local FBs
THIS^.CallFBs();
END_METHOD

METHOD PROTECTED CallFBs : BOOL
_Axis.ReadStatus();

(* MC_Power *)
MCPower(Axis := _Axis, Enable_Positive := NOT _InhibitFeedPositive, Enable_Negative := NOT _InhibitFeedNegative);
IF MCPower.Error THEN
    _Error   := TRUE;
    _ErrorID := MCPower.ErrorID;
END_IF

(* MC_MoveAbsolute *)
RingBuffer_MCMoveAbsolute(Axis := _Axis);
IF (MCMoveAbsolute <> 0) AND_THEN NOT MCMoveAbsolute^.Busy THEN
    IF MCMoveAbsolute^.Error THEN
        _Error   := TRUE;
        _ErrorID := MCMoveAbsolute^.ErrorID;
    ELSE
        MCMoveAbsolute^(Axis := _Axis, Execute := FALSE);
    END_IF
END_IF

(* MC_MoveRelative *)
RingBuffer_MCMoveRelative(Axis := _Axis);
IF (MCMoveRelative <> 0) AND_THEN NOT MCMoveRelative^.Busy THEN
    IF MCMoveRelative^.Error THEN
        _Error   := TRUE;
        _ErrorID := MCMoveRelative^.ErrorID;
    ELSE
        MCMoveRelative^(Axis := _Axis, Execute := FALSE);
    END_IF
END_IF

(* MC_MoveVelocity *)
RingBuffer_MCMoveVelocity(Axis := _Axis);
IF (MCMoveVelocity <> 0) AND_THEN ((NOT MCMoveVelocity^.Busy) OR MCMoveVelocity^.InVelocity) THEN
    IF MCMoveVelocity^.Error THEN
        _Error   := TRUE;
        _ErrorID := MCMoveVelocity^.ErrorID;
    ELSE
        MCMoveVelocity^(Axis := _Axis, Execute := FALSE);
    END_IF
END_IF

(* MC_MoveModulo *)
RingBuffer_MCMoveModulo(Axis := _Axis);
IF (MCMoveModulo <> 0) AND_THEN NOT MCMoveModulo^.Busy THEN
    IF MCMoveModulo^.Error THEN
        _Error   := TRUE;
        _ErrorID := MCMoveModulo^.ErrorID;
    ELSE
        MCMoveModulo^(Axis := _Axis, Execute := FALSE);
    END_IF
END_IF

//(* MC_MoveSuperimposed *)
//MCMoveSuperimposed(
//	Axis:= _Axis,
//	ActualVelocityDiff =>_ActualSuperPosVeloDiff,
//	ActualDistance =>_ActualSuperPosDistance,
//	ActualLength =>_ActualSuperPosLength,
//	ActualAcceleration =>_ActualSuperPosAccel,
//	ActualDeceleration =>_ActualSuperPosDecel,
//	CommandAborted =>_SuperPosAborted,
//	Done =>_SuperPosDone,
//	Busy =>_SuperPosBusy);
//IF NOT MCMoveSuperimposed.Busy THEN
//	IF MCMoveSuperimposed.Error THEN
//		_Error   := TRUE;
//		_ErrorID := MCMoveSuperimposed.ErrorID;
//	END_IF
//	IF MCMoveSuperimposed.Warning THEN
//		_Warning   := TRUE;
//		_WarningID := MCMoveSuperimposed.WarningId;
//	END_IF
//	MCMoveSuperimposed(
//		Execute:= FALSE,
//		Axis:= _Axis);
//END_IF

//(* MC_AbortSuperposition *)
//MCAbortSuperposition(
//	Axis:= _Axis);
//IF NOT MCAbortSuperposition.Busy THEN
//    IF MCAbortSuperposition.Error THEN
//        _Error   := TRUE;
//        _ErrorID := MCAbortSuperposition.ErrorID;
//    END_IF
//	MCAbortSuperposition(
//		Execute:= FALSE, 
//		Axis:= _Axis);
//END_IF

(*MC_Jog*)
MCJog(Axis := _Axis);
IF MCJog.Error THEN
    _Error   := TRUE;
    _ErrorID := MCJog.ErrorID;
END_IF

(* MC_MoveHalt *)
MCHalt(Axis := _Axis);
IF NOT MCHalt.Busy THEN
    IF MCHalt.Error THEN
        _Error   := TRUE;
        _ErrorID := MCHalt.ErrorID;
    ELSE
        MCHalt(Axis := _Axis, Execute := FALSE);
    END_IF
END_IF

(* FB_HomeRoutine_SetZeroHere *)
IF ipHomeMethod <> 0 AND_THEN ipHomeMethod.Axis <> 0 THEN
    ipHomeMethod.CyclicLogic();
    IF NOT ipHomeMethod.Busy THEN
        IF ipHomeMethod.Error AND NOT HomePreviouslyErrored THEN
            //This is used to trap circular errors (I_MotionStratery resets error bit on next execute)
            HomePreviouslyErrored := TRUE;
            _Error                := TRUE;
            _ErrorID              := ipHomeMethod.ErrorID;
        END_IF
    END_IF
END_IF

(* FB_ResetRoutine_CoEDrive *)
IF ipResetMethod <> 0 AND_THEN ipResetMethod.Axis <> 0 THEN
    ipResetMethod.CyclicLogic();
    IF NOT ipResetMethod.Busy AND NOT ResetPreviouslyErrored THEN
        IF ipResetMethod.Error THEN
            //This is used to trap circular errors (I_MotionStratery resets error bit on next execute)
            ResetPreviouslyErrored := TRUE;
            _Error                 := TRUE;
            _ErrorID               := ipResetMethod.ErrorID;
        END_IF
    END_IF
END_IF

(* MC_WriteParameterPersistent *)
MCWriteParameter(Axis := _Axis);
IF NOT MCWriteParameter.Busy THEN
    IF MCWriteParameter.Error THEN
        _Error   := TRUE;
        _ErrorID := MCWriteParameter.ErrorID;
    ELSE
        MCWriteParameter(Axis := _Axis, Execute := FALSE);
    END_IF
END_IF

(* MC_WriteBoolParameterPersistent *)
MCWriteBoolParameter(Axis := _Axis);
IF NOT MCWriteBoolParameter.Busy THEN
    IF MCWriteBoolParameter.Error THEN
        _Error   := TRUE;
        _ErrorID := MCWriteBoolParameter.ErrorID;
    ELSE
        MCWriteBoolParameter(Axis := _Axis, Execute := FALSE);
    END_IF
END_IF

_Busy := ((MCMoveAbsolute <> 0) AND_THEN MCMoveAbsolute^.Busy) OR ((MCMoveRelative <> 0) AND_THEN MCMoveRelative^.Busy) OR ((MCMoveVelocity <> 0) AND_THEN MCMoveVelocity^.Busy) OR
         ((MCMoveModulo <> 0) AND_THEN MCMoveModulo^.Busy) OR MCJog.Busy OR MCHalt.Busy OR ((ipHomeMethod <> 0) AND_THEN ipHomeMethod.Busy) OR ((ipResetMethod <> 0) AND_THEN ipResetMethod.Busy) OR
         MCWriteParameter.Busy OR MCWriteBoolParameter.Busy;
END_METHOD

METHOD PROTECTED Initialize : BOOL
VAR_INST
    LinkMissing : BOOL;
END_VAR
// Verify that the AXIS_REF is actually linked with the NC
IF F_GetMappingStatus(ADR(_Axis.NcToPlc), SIZEOF(_Axis.NcToPlc)) <> EPlcMappingStatus.MS_Mapped THEN
    IF NOT Parameters_MotionControl.ALLOW_UNLINKED_NC_AXES THEN
        IF NOT LinkMissing THEN
            Trace('Axis is not linked to NC');
            LinkMissing := TRUE;
        END_IF

        RETURN;
    END_IF
END_IF

IF F_GetMappingStatus(ADR(_Axis.PlcToNc), SIZEOF(_Axis.PlcToNc)) <> EPlcMappingStatus.MS_Mapped THEN
    IF NOT Parameters_MotionControl.ALLOW_UNLINKED_NC_AXES THEN
        IF NOT LinkMissing THEN
            Trace('Axis is not linked to NC');
            LinkMissing := TRUE;
        END_IF

        RETURN;
    END_IF
END_IF

// AxisId will be populated by the NC when it finishes starting

// This prevents requesting motion before NC Init/nuisance errors
IF _Axis.NcToPlc.AxisId = 0 THEN
    IF NOT Parameters_MotionControl.ALLOW_UNLINKED_NC_AXES THEN
        RETURN;
    END_IF
END_IF

// Use default home and reset methods until they are set by parent
IF ipHomeMethod = 0 THEN
    THIS^.HomeMethod := DefaultHome;
END_IF

IF ipResetMethod = 0 THEN
    THIS^.ResetMethod := DefaultReset;
END_IF

// Read all NC parameters
IF Parameters_MotionControl.ALLOW_UNLINKED_NC_AXES THEN
    Initialize := TRUE;
ELSE
    MCReadParameterSet(Parameter := _AxisParameters, Axis := _Axis, Execute := TRUE);
    IF NOT MCReadParameterSet.Busy THEN
        IF MCReadParameterSet.Error THEN
            _Error   := TRUE;
            _ErrorID := MCReadParameterSet.ErrorID;
        ELSIF MCReadParameterSet.Done THEN
            _Velocity     := _AxisParameters.fVeloSlowManual;
            _Acceleration := _AxisParameters.fAcceleration;
            _Deceleration := _AxisParameters.fDeceleration;
            _Jerk         := _AxisParameters.fJerk;
            Trace('Axis initialization complete');
            Initialize := TRUE;
        END_IF

        MCReadParameterSet(Parameter := _AxisParameters, Axis := _Axis, Execute := FALSE);
    END_IF
END_IF
END_METHOD

PROPERTY AxisParameters : REFERENCE TO ST_AxisParameterSet
GET
AxisParameters REF= _AxisParameters;
END_GET
END_PROPERTY

END_FUNCTION_BLOCK

// Function Blocks/FB_RingBuffer_MCMoveAbsolute
FUNCTION_BLOCK FB_RingBuffer_MCMoveAbsolute
VAR_IN_OUT
    Axis : AXIS_REF;
END_VAR

VAR_OUTPUT
END_VAR

VAR
    MCMoveAbsoluteCA : ARRAY[0..1] OF MC_MoveAbsolute;
    _CurrentFB       : UDINT;
    i                : UDINT;
END_VAR

(* This buffer ensures you always have a clean FB to use for a move *)

FOR i := 0 TO 1 DO
    MCMoveAbsoluteCA[i](Axis := Axis);
END_FOR

PROPERTY CurrentFB : POINTER TO MC_MoveAbsolute
GET
CurrentFB := ADR(MCMoveAbsoluteCA[_CurrentFB]);
END_GET
END_PROPERTY

METHOD GetNewFB : POINTER TO MC_MoveAbsolute
VAR_INPUT
END_VAR
_CurrentFB := _CurrentFB + 1;
IF _CurrentFB > 1 THEN
    MCMoveAbsoluteCA[1].Execute := FALSE;
    _CurrentFB                  := 0;
ELSE
    MCMoveAbsoluteCA[_CurrentFB - 1].Execute := FALSE;
END_IF

GetNewFB := ADR(MCMoveAbsoluteCA[_CurrentFB]);
END_METHOD

END_FUNCTION_BLOCK

// Function Blocks/FB_RingBuffer_MCMoveRelative
FUNCTION_BLOCK FB_RingBuffer_MCMoveRelative
VAR_IN_OUT
    Axis : AXIS_REF;
END_VAR

VAR_OUTPUT
END_VAR

VAR
    MCMoveRelative : ARRAY[0..1] OF MC_MoveRelative;
    _CurrentFB     : UDINT;
    i              : UDINT;
END_VAR

(* This buffer ensures you always have a clean FB to use for a move *)

FOR i := 0 TO 1 DO
    MCMoveRelative[i](Axis := Axis);
END_FOR

PROPERTY CurrentFB : POINTER TO MC_MoveRelative
GET
CurrentFB := ADR(MCMoveRelative[_CurrentFB]);
END_GET
END_PROPERTY

METHOD GetNewFB : POINTER TO MC_MoveAbsolute
VAR_INPUT
END_VAR
_CurrentFB := _CurrentFB + 1;
IF _CurrentFB > 1 THEN
    MCMoveRelative[1].Execute := FALSE;
    _CurrentFB                := 0;
ELSE
    MCMoveRelative[_CurrentFB - 1].Execute := FALSE;
END_IF

GetNewFB := ADR(MCMoveRelative[_CurrentFB]);
END_METHOD

END_FUNCTION_BLOCK

// Function Blocks/FB_RingBuffer_MCMoveVelocity
FUNCTION_BLOCK FB_RingBuffer_MCMoveVelocity
VAR_IN_OUT
    Axis : AXIS_REF;
END_VAR

VAR_OUTPUT
END_VAR

VAR
    MCMoveVelocity : ARRAY[0..1] OF MC_MoveVelocity;
    _CurrentFB     : UDINT;
    i              : UDINT;
END_VAR

(* This buffer ensures you always have a clean FB to use for a move *)

FOR i := 0 TO 1 DO
    MCMoveVelocity[i](Axis := Axis);
END_FOR

PROPERTY CurrentFB : POINTER TO MC_MoveVelocity
GET
CurrentFB := ADR(MCMoveVelocity[_CurrentFB]);
END_GET
END_PROPERTY

METHOD GetNewFB : POINTER TO MC_MoveAbsolute
VAR_INPUT
END_VAR
_CurrentFB := _CurrentFB + 1;
IF _CurrentFB > 1 THEN
    MCMoveVelocity[1].Execute := FALSE;
    _CurrentFB                := 0;
ELSE
    MCMoveVelocity[_CurrentFB - 1].Execute := FALSE;
END_IF

GetNewFB := ADR(MCMoveVelocity[_CurrentFB]);
END_METHOD

END_FUNCTION_BLOCK

// Function Blocks/FB_RingBuffer_MCMoveModulo
FUNCTION_BLOCK FB_RingBuffer_MCMoveModulo
VAR_IN_OUT
    Axis : AXIS_REF;
END_VAR

VAR_OUTPUT
END_VAR

VAR
    MCMoveModulo : ARRAY[0..1] OF MC_MoveModulo;
    _CurrentFB   : UDINT;
    i            : UDINT;
END_VAR

(* This buffer ensures you always have a clean FB to use for a move *)

FOR i := 0 TO 1 DO
    MCMoveModulo[i](Axis := Axis);
END_FOR

PROPERTY CurrentFB : POINTER TO MC_MoveModulo
GET
CurrentFB := ADR(MCMoveModulo[_CurrentFB]);
END_GET
END_PROPERTY

METHOD GetNewFB : POINTER TO MC_MoveAbsolute
VAR_INPUT
END_VAR
_CurrentFB := _CurrentFB + 1;
IF _CurrentFB > 1 THEN
    MCMoveModulo[1].Execute := FALSE;
    _CurrentFB              := 0;
ELSE
    MCMoveModulo[_CurrentFB - 1].Execute := FALSE;
END_IF

GetNewFB := ADR(MCMoveModulo[_CurrentFB]);
END_METHOD

END_FUNCTION_BLOCK

// Function Blocks/FB_BasicSlaveAxis
FUNCTION_BLOCK FB_BasicSlaveAxis EXTENDS FB_BasicAxis IMPLEMENTS I_BasicSlaveAxis
VAR
    MCGearInMultimaster : MC_GearInMultiMaster;
    MCGearOut           : MC_GearOut;
    {attribute 'hide'}
    DummyAxis     : AXIS_REF;
    _Master1      : REFERENCE TO AXIS_REF;
    _Master2      : REFERENCE TO AXIS_REF;
    _Master3      : REFERENCE TO AXIS_REF;
    _Master4      : REFERENCE TO AXIS_REF;
    _RatioMaster1 : LREAL := 1;
    _RatioMaster2 : LREAL := 1;
    _RatioMaster3 : LREAL := 1;
    _RatioMaster4 : LREAL := 1;
END_VAR

//There should be no code in the function block body

METHOD Home : BOOL
IF _Busy OR _Error OR ipHomeMethod = 0 THEN
    RETURN;
END_IF

MCGearInMultimaster(Slave := _Axis, Enable := FALSE);
Home := SUPER^.Home();
END_METHOD

METHOD MoveAbsolute : BOOL
VAR_INPUT
    Position      : LREAL;
    AbortPrevious : BOOL;
END_VAR
IF _Error THEN
    RETURN;
ELSE
    IF (_Busy AND NOT AbortPrevious) THEN
        RETURN;
    END_IF
END_IF

MCGearInMultimaster(Slave := _Axis, Enable := FALSE);
MoveAbsolute := SUPER^.MoveAbsolute(Position, AbortPrevious);
END_METHOD

METHOD MoveModulo : BOOL
VAR_INPUT
    Position      : LREAL;
    Direction     : MC_Direction;
    AbortPrevious : BOOL;
END_VAR
IF _Error THEN
    RETURN;
ELSE
    IF (_Busy AND NOT AbortPrevious) THEN
        RETURN;
    END_IF
END_IF

MCGearInMultimaster(Slave := _Axis, Enable := FALSE);
MoveModulo := SUPER^.MoveModulo(Position, Direction, AbortPrevious);
END_METHOD

METHOD MoveRelative : BOOL
VAR_INPUT
    Distance      : LREAL;
    AbortPrevious : BOOL;
END_VAR
IF _Error THEN
    RETURN;
ELSE
    IF (_Busy AND NOT AbortPrevious) THEN
        RETURN;
    END_IF
END_IF

MCGearInMultimaster(Slave := _Axis, Enable := FALSE);
MoveRelative := SUPER^.MoveRelative(Distance, AbortPrevious);
END_METHOD

METHOD MoveVelocity : BOOL
VAR_INPUT
    Velocity      : LREAL;
    AbortPrevious : BOOL;
END_VAR
IF _Error THEN
    RETURN;
ELSE
    IF (_Busy AND NOT AbortPrevious) THEN
        RETURN;
    END_IF
END_IF

MCGearInMultimaster(Slave := _Axis, Enable := FALSE);
MoveVelocity := SUPER^.MoveVelocity(Velocity, AbortPrevious);
END_METHOD

METHOD Reset : BOOL
IF _Axis.Status.Coupled AND NOT _Axis.Status.Error THEN
    //Allow this method to be called and reset flags if axis was reset through master
    _Error   := FALSE;
    _ErrorID := 0;
    Reset    := TRUE;
    RETURN;
ELSIF _Busy OR _Axis.Status.Coupled OR ipResetMethod = 0 THEN
    //If axis is coupled it should be reset through the master
    RETURN;
END_IF

IF SUPER^.Reset() THEN
    Reset := TRUE;
END_IF

//IF ipResetMethod.Execute() THEN

//    _Error   := FALSE;

//    _ErrorID := 0;

//    Reset    := TRUE;

//END_IF
END_METHOD

METHOD PUBLIC GearIn : BOOL
VAR_INPUT
END_VAR
IF _Busy OR _Error THEN
    RETURN;
END_IF

MCGearInMultimaster(Master1      := _Master1,
                    Master2      := _Master2,
                    Master3      := _Master3,
                    Master4      := _Master4,
                    Slave        := _Axis,
                    Enable       := TRUE,
                    GearRatio1   := _RatioMaster1,
                    GearRatio2   := _RatioMaster2,
                    GearRatio3   := _RatioMaster3,
                    GearRatio4   := _RatioMaster4,
                    Acceleration := _Acceleration,
                    Deceleration := _Deceleration,
                    Jerk         := _Jerk);

GearIn := TRUE;
END_METHOD

METHOD GearOut : BOOL
IF _Busy THEN
    RETURN;
END_IF

MCGearInMultimaster(Master1      := _Master1,
                    Master2      := _Master2,
                    Master3      := _Master3,
                    Master4      := _Master4,
                    Slave        := _Axis,
                    Enable       := FALSE,
                    GearRatio1   := _RatioMaster1,
                    GearRatio2   := _RatioMaster2,
                    GearRatio3   := _RatioMaster3,
                    GearRatio4   := _RatioMaster4,
                    Acceleration := _Acceleration,
                    Deceleration := _Deceleration,
                    Jerk         := _Jerk);

MCGearOut(Slave := _Axis, Execute := TRUE);
GearOut := TRUE;
END_METHOD

PROPERTY InGear : BOOL
GET
InGear := MCGearInMultimaster.InGear;
END_GET
END_PROPERTY

PROPERTY Master1 : REFERENCE TO AXIS_REF
GET
IF __ISVALIDREF(_Master1) THEN
    Master1 REF= _Master1;
END_IF
END_GET
SET
_Master1 REF= Master1;
END_SET
END_PROPERTY

PROPERTY Master2 : REFERENCE TO AXIS_REF
GET
IF __ISVALIDREF(_Master2) THEN
    Master2 REF= _Master2;
END_IF
END_GET
SET
_Master2 REF= Master2;
END_SET
END_PROPERTY

PROPERTY Master3 : REFERENCE TO AXIS_REF
GET
IF __ISVALIDREF(_Master3) THEN
    Master3 REF= _Master3;
END_IF
END_GET
SET
_Master3 REF= Master3;
END_SET
END_PROPERTY

PROPERTY Master4 : REFERENCE TO AXIS_REF
GET
IF __ISVALIDREF(_Master4) THEN
    Master4 REF= _Master4;
END_IF
END_GET
SET
_Master4 REF= Master4;
END_SET
END_PROPERTY

PROPERTY RatioMaster1 : LREAL
GET
RatioMaster1 := _RatioMaster1;
END_GET
SET
_RatioMaster1 := RatioMaster1;
END_SET
END_PROPERTY

PROPERTY RatioMaster2 : LREAL
GET
RatioMaster2 := _RatioMaster2;
END_GET
SET
_RatioMaster2 := RatioMaster2;
END_SET
END_PROPERTY

PROPERTY RatioMaster3 : LREAL
GET
RatioMaster3 := _RatioMaster3;
END_GET
SET
_RatioMaster3 := RatioMaster3;
END_SET
END_PROPERTY

PROPERTY RatioMaster4 : LREAL
GET
RatioMaster4 := _RatioMaster4;
END_GET
SET
_RatioMaster4 := RatioMaster4;
END_SET
END_PROPERTY

METHOD Stop : BOOL
MCGearInMultimaster(Slave := _Axis, Enable := FALSE);
IF SUPER^.Stop() THEN
    Stop := TRUE;
END_IF
END_METHOD

METHOD PUBLIC CyclicLogic
VAR_INPUT
END_VAR
IF NOT _InitComplete THEN
    _InitComplete := THIS^.Initialize();
    RETURN;
END_IF

//Call local FBs
SUPER^.CyclicLogic();
END_METHOD

METHOD PROTECTED CallFBs : BOOL
VAR_INPUT
END_VAR
SUPER^.CallFBs();

(* MC_GearInMultimaster *)
MCGearInMultimaster(Slave        := _Axis,
                    GearRatio1   := _RatioMaster1,
                    GearRatio2   := _RatioMaster2,
                    GearRatio3   := _RatioMaster3,
                    GearRatio4   := _RatioMaster4,
                    Acceleration := _Acceleration,
                    Deceleration := _Deceleration,
                    Jerk         := _Jerk);

//IF NOT MCGearInMultimaster.Busy THEN
IF MCGearInMultimaster.Error THEN
    _Error   := TRUE;
    _ErrorID := MCGearInMultimaster.ErrorID;
END_IF

//	MCGearInMultimaster(Slave := _Axis,Enable:= FALSE);

//END_IF

(* MC_GearOut *)
MCGearOut(Slave := _Axis);
IF NOT MCGearOut.Busy THEN
    IF MCGearOut.Error THEN
        _Error   := TRUE;
        _ErrorID := MCGearOut.ErrorID;
    END_IF

    MCGearOut(Slave := _Axis, Execute := FALSE);
END_IF

_Busy := _Busy OR MCGearOut.Error;
END_METHOD

METHOD PROTECTED Initialize : BOOL
VAR_INPUT
END_VAR
_Master1   REF= DummyAxis;
_Master2   REF= DummyAxis;
_Master3   REF= DummyAxis;
_Master4   REF= DummyAxis;
Initialize := SUPER^.Initialize();
END_METHOD

END_FUNCTION_BLOCK

// Interfaces/I_BasicSlaveAxis
INTERFACE I_BasicSlaveAxis EXTENDS I_BasicAxis

METHOD PUBLIC GearIn : BOOL
VAR_INPUT
END_VAR
END_METHOD

METHOD GearOut : BOOL
END_METHOD

PROPERTY InGear : BOOL
GET
END_GET
END_PROPERTY

PROPERTY Master1 : REFERENCE TO AXIS_REF
GET
END_GET
SET
END_SET
END_PROPERTY

PROPERTY Master2 : REFERENCE TO AXIS_REF
GET
END_GET
SET
END_SET
END_PROPERTY

PROPERTY Master3 : REFERENCE TO AXIS_REF
GET
END_GET
SET
END_SET
END_PROPERTY

PROPERTY Master4 : REFERENCE TO AXIS_REF
GET
END_GET
SET
END_SET
END_PROPERTY

PROPERTY RatioMaster1 : LREAL
GET
END_GET
SET
END_SET
END_PROPERTY

PROPERTY RatioMaster2 : LREAL
GET
END_GET
SET
END_SET
END_PROPERTY

PROPERTY RatioMaster3 : LREAL
GET
END_GET
SET
END_SET
END_PROPERTY

PROPERTY RatioMaster4 : LREAL
GET
END_GET
SET
END_SET
END_PROPERTY

END_INTERFACE

// Function Blocks/FB_CamSlaveAxis
FUNCTION_BLOCK FB_CamSlaveAxis EXTENDS FB_BasicAxis IMPLEMENTS I_CamSlaveAxis
VAR
    {attribute 'hide'}
    DummyAxis                   : AXIS_REF;
    SequenceState               : UDINT;
    MCCamOut                    : MC_CamOut;
    MCCamIn                     : MC_CamIn;
    MCCamTableSelect            : MC_CamTableSelect;
    MCSetCamOnlineChangeMode    : MC_SetCamOnlineChangeMode;
    MCWriteMotionFunction       : MC_WriteMotionFunction;
    MCReadCamTableSlaveDynamics : MC_ReadCamTableSlaveDynamics;
    MasterParameters            : ST_AxisParameterSet; // Master Information 
    InWindow                    : BOOL;
    SemaphoreBusy               : BOOL;
    MoveTarget                  : LREAL;
    OldTableSelect              : UDINT;
    CurrentTableSelect          : UDINT := 1;
    CurrentPoints               : ARRAY[1..Parameters_MotionControl.CAM_SLAVE_AXIS_MAX_CAM_POINTS] OF MC_MotionFunctionPoint;
    CurrentTable                : MC_Cam_Ref;
    ReadSlaveDynamicsMasterPos  : LREAL;
    MoveModuloDirection         : MC_Direction;
    FindSlavePositionCommand    : BOOL; // Report Slave's Sync Position Based On Specified Master Position
    FindSyncPositionCommand     : BOOL; // Report Slave's Sync Position Based On Set Master Position 
    StartSyncCommand            : BOOL; // execute sync move if required and couple slave to master using cam table
    StartCoupleCommand          : BOOL; // couple slave to master using cam table, no sync move used
    UpdateTableCommand          : BOOL; // Update Current Cam Table
    ChangeModeCommand           : BOOL; // Update OnLineChangeMode 
    FindDone                    : BOOL; // indicates slave position lookup is complete and _SyncPos is updated
    SequenceError               : BOOL;
    SequenceErrorID             : UDINT;
    ReadyToCam                  : BOOL;
    _CamParameters              : REFERENCE TO ST_CamParameters; // Parameters for Camming Motion	
    _InSync                     : BOOL;                          // indicates slave is coupled	
    _Master                     : REFERENCE TO AXIS_REF;
    _RunningTable               : UDINT; // indicates running cam table in parameter array
    _SyncPos                    : LREAL; // indicates cam table slave position for designated master position
END_VAR

//There should be no code in the function block body

METHOD Home : BOOL
IF _Busy OR _Error OR ipHomeMethod = 0 THEN
    RETURN;
END_IF

SequenceState := 0;
Home          := SUPER^.Home();
END_METHOD

METHOD MoveModulo : BOOL
VAR_INPUT
    Position      : LREAL;
    Direction     : MC_Direction;
    AbortPrevious : BOOL;
END_VAR
IF _Error THEN
    RETURN;
ELSE
    IF (_Busy AND NOT StartSyncCommand) THEN
        RETURN;
    END_IF
END_IF

MoveModulo := SUPER^.MoveModulo(Position, Direction, AbortPrevious);
END_METHOD

METHOD Reset : BOOL
IF _Busy OR _Axis.Status.Coupled OR ipResetMethod = 0 THEN
    //If axis is coupled it should be reset through the master
    RETURN;
END_IF

IF SUPER^.Reset() THEN
    IF SequenceError THEN
        SequenceError   := FALSE;
        SequenceErrorID := 0;
        SequenceState   := E_CamAxisState.eCamAxisState_Disabled;
    END_IF

    IF MCReadCamTableSlaveDynamics.Error THEN
        MCReadCamTableSlaveDynamics(Execute := FALSE);
    END_IF

    IF __ISVALIDREF(_Master) THEN
        IF MCCamTableSelect.Error THEN
            MCCamTableSelect(Master   := _Master,
                             Slave    := _Axis,
                             CamTable := CurrentTable,
                             Execute  := FALSE);
        END_IF

        IF MCCamIn.Error THEN
            McCamIn(Master := _Master, Slave := _Axis, Execute := FALSE);
        END_IF

        IF MCCamOut.Error THEN
            McCamOut(Slave := _Axis, Execute := FALSE);
        END_IF
    END_IF

    IF MCWriteMotionFunction.Error THEN
        MCWriteMotionFunction(Execute := FALSE);
    END_IF

    IF MCSetCamOnlineChangeMode.Error THEN
        MCSetCamOnlineChangeMode(Execute := FALSE);
    END_IF

    Reset := TRUE;
END_IF
END_METHOD

METHOD Stop : BOOL
//StopCommand := TRUE;

//Stop                 := TRUE;
Stop := SUPER^.Stop();
END_METHOD

PROPERTY CamParameters : REFERENCE TO ST_CamParameters
GET
IF __ISVALIDREF(_CamParameters) THEN
    CamParameters REF= _CamParameters;
END_IF
END_GET
SET
_CamParameters REF= CamParameters;
END_SET
END_PROPERTY

METHOD ChangeMode : BOOL
VAR_INPUT
END_VAR
IF _Error OR _Busy OR NOT ReadyToCam THEN
    RETURN;
ELSE
    ChangeModeCommand := TRUE;
    ChangeMode        := TRUE;
END_IF
END_METHOD

METHOD FindSlavePos : BOOL
VAR_INPUT
END_VAR
IF _Error OR _Busy OR NOT ReadyToCam THEN
    RETURN;
ELSE
    FindSlavePositionCommand := TRUE;
    FindSlavePos             := TRUE;
END_IF
END_METHOD

METHOD FindSyncPos : BOOL
VAR_INPUT
END_VAR
IF _Error OR _Busy OR NOT ReadyToCam THEN
    RETURN;
ELSE
    FindSyncPositionCommand := TRUE;
    FindSyncPos             := TRUE;
END_IF
END_METHOD

PROPERTY InSync : BOOL
GET
InSync := _InSync;
END_GET
END_PROPERTY

PROPERTY Master : REFERENCE TO Tc2_MC2.AXIS_REF
GET
IF __ISVALIDREF(_Master) THEN
    Master REF= _Master;
END_IF
END_GET
SET
_Master REF= Master;
END_SET
END_PROPERTY

PROPERTY RunningTable : UDINT
GET
RunningTable := _RunningTable;
END_GET
END_PROPERTY

METHOD StartCouple : BOOL
VAR_INPUT
END_VAR
IF _Error OR _Busy OR NOT ReadyToCam OR NOT FindDone THEN
    RETURN;
ELSE
    StartCoupleCommand := TRUE;
    StartCouple        := TRUE;
END_IF
END_METHOD

METHOD StartSync : BOOL
VAR_INPUT
END_VAR
IF _Error OR _Busy OR NOT ReadyToCam OR _InSync THEN
    RETURN;
ELSE
    StartSyncCommand := TRUE;
    StartSync        := TRUE;
END_IF
END_METHOD

PROPERTY SyncPos : LREAL
GET
SyncPos := _SyncPos;
END_GET
END_PROPERTY

METHOD UpdateTable : BOOL
VAR_INPUT
END_VAR
IF _Error OR _Busy OR NOT ReadyToCam THEN
    RETURN;
ELSE
    UpdateTableCommand := TRUE;
    UpdateTable        := TRUE;
END_IF
END_METHOD

METHOD PUBLIC CyclicLogic
IF NOT _InitComplete THEN
    _InitComplete := THIS^.Initialize();
    RETURN;
END_IF

_InSync    := _Axis.Status.Coupled;
ReadyToCam :=
    __ISVALIDREF(_CamParameters) AND __ISVALIDREF(_Master) AND_THEN (_Master.NcToPlc.AxisId > 0) AND_THEN (_Axis.NcToPlc.AxisId > 0) AND_THEN (_Master.NcToPlc.AxisId <> _Axis.NcToPlc.AxisId);

IF _Axis.Status.Error THEN
    SequenceState := E_CamAxisState.eCamAxisState_Disabled;
END_IF

CASE SequenceState OF
    E_CamAxisState.eCamAxisState_Disabled:
        // Reset Outputs 
        SequenceError := FALSE;
        FindDone      := FALSE;
        _RunningTable := 0;
        _SyncPos      := 0.0;

        // Reset Semaphore Inputs 
        FindSlavePositionCommand := FALSE;
        FindSyncPositionCommand  := FALSE;
        StartSyncCommand         := FALSE;
        StartCoupleCommand       := FALSE;
        UpdateTableCommand       := FALSE;
        ChangeModeCommand        := FALSE;
        SequenceErrorID          := 0;

        // Reset All Function Block Calls 
        MCCamTableSelect.Execute            := FALSE;
        MCReadCamTableSlaveDynamics.Execute := FALSE;
        McCamIn.Execute                     := FALSE;
        McCamOut.Execute                    := FALSE;
        MCSetCamOnlineChangeMode.Execute    := FALSE;
        McWriteMotionFunction.Execute       := FALSE;

        // Wait for Function Block Enable 
        IF NOT _Axis.Status.Error AND ReadyToCam THEN
            // Function Block Has to Be Enabled and Slave Axis is Error Free Before Continue 
            SequenceState := E_CamAxisState.eCamAxisState_ReadMasterParameters;
        END_IF
    E_CamAxisState.eCamAxisState_ReadMasterParameters:
        MCReadParameterSet(Execute := TRUE, Parameter := MasterParameters, Axis := _Master);
        IF MCReadParameterSet.Error THEN
            //MCReadParameterSet(Execute := FALSE, Parameter := MasterParameters, Axis := _Master);
            SequenceErrorID := MCReadParameterSet.ErrorID;
            SequenceState   := E_CamAxisState.eCamAxisState_Error;
        ELSIF MCReadParameterSet.Done THEN
            MCReadParameterSet(Execute := FALSE, Parameter := MasterParameters, Axis := _Master);
            SequenceState := E_CamAxisState.eCamAxisState_AxisInitDone;
        END_IF
    E_CamAxisState.eCamAxisState_ReadSlaveParameters:
        MCReadParameterSet(Execute := TRUE, Parameter := _AxisParameters, Axis := _Axis);
        IF MCReadParameterSet.Error THEN
            //MCReadParameterSet(Execute := FALSE, Parameter := _AxisParameters, Axis := _Axis);
            SequenceErrorID := MCReadParameterSet.ErrorID;
            SequenceState   := E_CamAxisState.eCamAxisState_Error;
        ELSIF MCReadParameterSet.Done THEN
            MCReadParameterSet(Execute := FALSE, Parameter := _AxisParameters, Axis := _Axis);
            SequenceState := E_CamAxisState.eCamAxisState_AxisInitDone;
        END_IF
    E_CamAxisState.eCamAxisState_AxisInitDone:
        // Inputs Should Be Off After Initialization or After An Error 
        IF NOT FindSlavePositionCommand AND NOT FindSyncPositionCommand AND NOT StartSyncCommand AND NOT StartCoupleCommand AND NOT UpdateTableCommand THEN
            SequenceState := E_CamAxisState.eCamAxisState_WaitForCommand;
        ELSE
            SequenceState := E_CamAxisState.eCamAxisState_Error;
        END_IF
    E_CamAxisState.eCamAxisState_WaitForCommand:
        IF FindSlavePositionCommand OR FindSyncPositionCommand OR StartSyncCommand THEN
            FindDone := FALSE;

            // DeCouple Slave If Coupled 
            IF _InSync THEN
                SequenceState := E_CamAxisState.eCamAxisState_DecoupleBeforeStart;
            ELSE
                SequenceState := E_CamAxisState.eCamAxisState_CheckTableSelect;
            END_IF
        ELSIF StartCoupleCommand AND FindDone THEN
            SequenceState := E_CamAxisState.eCamAxisState_CoupleSlave;
        ELSIF ChangeModeCommand THEN
            // Can't Change Table Yet Because We Don't Have a Cam Table ID 

            // Update OnLineChangeMode 
            SequenceState := E_CamAxisState.eCamAxisState_SetChangeMode;
        END_IF
    E_CamAxisState.eCamAxisState_DecoupleBeforeStart:
        McCamOut.Execute := TRUE;
        IF NOT McCamOut.BUSY THEN
            IF McCamOut.ERROR THEN
                SequenceErrorID := McCamOut.ERRORID;
                SequenceState   := E_CamAxisState.eCamAxisState_Error;
            ELSE
                McCamOut.Execute := FALSE;
                SequenceState    := E_CamAxisState.eCamAxisState_CheckTableSelect;
            END_IF
        END_IF
    E_CamAxisState.eCamAxisState_CheckTableSelect:
        IF _CamParameters.TableSelect < 1 OR _CamParameters.TableSelect > Parameters_MotionControl.CAM_SLAVE_AXIS_TABLES THEN
            SequenceState := E_CamAxisState.eCamAxisState_Error;
        ELSE
            SequenceState := E_CamAxisState.eCamAxisState_LoadCamTable;
        END_IF
    E_CamAxisState.eCamAxisState_LoadCamTable:
        // Lock The Selected Table Number In Case User Changes It During Processesing 
        CurrentTableSelect := _CamParameters.TableSelect;
        CurrentPoints      := _CamParameters.CamTable[CurrentTableSelect].Points;
        OldTableSelect     := CurrentTableSelect;

        // Configure Cam Reference 
        CurrentTable.pArray      := ADR(CurrentPoints);
        CurrentTable.ArraySize   := SIZEOF(CurrentPoints);
        CurrentTable.NoOfColumns := 1; // Always 1 for Motion Functions 
        CurrentTable.NoOfRows    := DINT_TO_UDINT(_CamParameters.CamTable[CurrentTableSelect].NumberOfPoints);
        CurrentTable.TableType   := MC_TABLETYPE_MOTIONFUNCTION;
        MCCamTableSelect.Execute := TRUE;
        IF MCCamTableSelect.Error THEN
            //MCCamTableSelect.Execute := FALSE;
            SequenceErrorID := MCCamTableSelect.ErrorID;
            SequenceState   := E_CamAxisState.eCamAxisState_Error;
        ELSIF MCCamTableSelect.Done THEN
            MCCamTableSelect.Execute := FALSE;
            SequenceState            := E_CamAxisState.eCamAxisState_CheckAxisStatus;
        END_IF
    E_CamAxisState.eCamAxisState_CheckAxisStatus:
        IF _Master.Status.Error THEN
            // Master Axis Has An Error (31 = Axis Fault) 
            SequenceState := E_CamAxisState.eCamAxisState_Error;
        ELSIF NOT _Axis.Status.ControlLoopClosed THEN // 20 = Control Loop Closed 

            // Slave Axis Is Not Enabled 
            SequenceState := E_CamAxisState.eCamAxisState_Error;
        ELSIF NOT _Master.Status.ControlLoopClosed AND (MasterParameters.nAxisType = 1 OR MasterParameters.nAxisType = 3) THEN
            // Master Axis Is Not Enabled 
            SequenceState := E_CamAxisState.eCamAxisState_Error;
        ELSE
            // Find Where Slave Axis Is Suppose To Be 
            IF FindSlavePositionCommand THEN
                // Report Slave's Sync Position Based On Specified Master Position 
                ReadSlaveDynamicsMasterPos := _CamParameters.MasterPos;
                SequenceState              := E_CamAxisState.eCamAxisState_ReadSlaveDynamics;
            ELSIF FindSyncPositionCommand OR StartSyncCommand THEN
                // Report Slave's Sync Position Based On Set Master Position 
                ReadSlaveDynamicsMasterPos := _Master.NcToPlc.ActPos;
                SequenceState              := E_CamAxisState.eCamAxisState_ReadSlaveDynamics;
            ELSE
                // User Must Have Reset Inputs 
                SequenceState := E_CamAxisState.eCamAxisState_WaitForCommand;
            END_IF
        END_IF
    E_CamAxisState.eCamAxisState_ReadSlaveDynamics:
        MCReadCamTableSlaveDynamics.Execute := TRUE;
        IF MCReadCamTableSlaveDynamics.Error THEN
            //MCReadCamTableSlaveDynamics.Execute := FALSE;
            SequenceErrorID := MCReadCamTableSlaveDynamics.ErrorID;
            SequenceState   := E_CamAxisState.eCamAxisState_Error;
        ELSIF MCReadCamTableSlaveDynamics.Done THEN
            _SyncPos                            := MCReadCamTableSlaveDynamics.SlavePosition + _CamParameters.SlaveOffset;
            MCReadCamTableSlaveDynamics.Execute := FALSE;
            FindDone                            := TRUE;
            FindSlavePositionCommand            := FALSE;
            FindSyncPositionCommand             := FALSE;
            IF StartSyncCommand THEN
                SequenceState := E_CamAxisState.eCamAxisState_DetermineSyncMove;
            ELSE
                SequenceState := E_CamAxisState.eCamAxisState_WaitForCommand;
            END_IF
        END_IF
    E_CamAxisState.eCamAxisState_DetermineSyncMove:
        // If You Need to Perform a Sync Move Other Than Mode Module Then Use Inputs _FindSlave or _FindSync To Find Sync Position, Perform Move 

        // Outside of This Function Block, Then Couple Using Input _StartCouple 
        IF ABS(_Axis.NcToPlc.ModuloActPos - MODABS(MCReadCamTableSlaveDynamics.SlavePosition + _CamParameters.SlaveOffset, _AxisParameters.fEncModuloFactor)) < ABS(_CamParameters.SyncWindow) THEN
            InWindow := TRUE;
        ELSE
            InWindow := FALSE;
        END_IF

        CASE _CamParameters.SyncMode OF
            E_CamSyncMode.eCamSyncMode_ShortestWay:
                // Move the Shortest Distance 
                MoveModuloDirection := MC_Shortest_Way;
                SequenceState       := E_CamAxisState.eCamAxisState_SlaveSyncMove;
            E_CamSyncMode.eCamSyncMode_Forward:
                // Move Only in the Forward Direction 
                MoveModuloDirection := MC_Positive_Direction;
                SequenceState       := E_CamAxisState.eCamAxisState_SlaveSyncMove;
            E_CamSyncMode.eCamSyncMode_Reverse:
                // Move Only in the Reverse Direction 
                MoveModuloDirection := MC_Negative_Direction;
                SequenceState       := E_CamAxisState.eCamAxisState_SlaveSyncMove;
            E_CamSyncMode.eCamSyncMode_Window_Forward:
                // Move Shortest Distance If In Window Else Move Forward 
                IF InWindow THEN
                    MoveModuloDirection := MC_Shortest_Way;
                ELSE
                    MoveModuloDirection := MC_Positive_Direction;
                END_IF

                SequenceState := E_CamAxisState.eCamAxisState_SlaveSyncMove;
            E_CamSyncMode.eCamSyncMode_Window_Reverse:
                // Move Shortest Distance If In Window Else Move Reverse 
                IF InWindow THEN
                    MoveModuloDirection := MC_Shortest_Way;
                ELSE
                    MoveModuloDirection := MC_Negative_Direction;
                END_IF

                SequenceState := E_CamAxisState.eCamAxisState_SlaveSyncMove;
        ELSE
            SequenceState := E_CamAxisState.eCamAxisState_Error;
        END_CASE
    E_CamAxisState.eCamAxisState_SlaveSyncMove:
        Velocity     := _CamParameters.SyncVelocity;
        Acceleration := _CamParameters.SyncAccel;
        Deceleration := _CamParameters.SyncDecel;
        Jerk         := _CamParameters.SyncJerk;
        MoveTarget   := MODABS(MCReadCamTableSlaveDynamics.SlavePosition + _CamParameters.SlaveOffset, _AxisParameters.fEncModuloFactor);
        SUPER^.MoveModulo(Position := MoveTarget, Direction := MoveModuloDirection, AbortPrevious := TRUE);
        IF SUPER^.MCMoveModulo^.Error THEN
            SequenceErrorID := SUPER^.MCMoveModulo^.ErrorID;
            SequenceState   := E_CamAxisState.eCamAxisState_Error;
        ELSIF SUPER^.MCMoveModulo^.Done THEN
            SequenceState := E_CamAxisState.eCamAxisState_CoupleSlave;
        END_IF
    E_CamAxisState.eCamAxisState_CoupleSlave:
        // MC_CamIn 
        McCamIn.Execute := TRUE;
        IF McCamIn.Error THEN
            StartSyncCommand := FALSE;

            //McCamIn.Execute  := FALSE;
            SequenceErrorID := McCamIn.ErrorID;
            SequenceState   := E_CamAxisState.eCamAxisState_Error;
        ELSIF McCamIn.CommandAborted THEN
            StartSyncCommand := FALSE;
            McCamIn.Execute  := FALSE;
            SequenceState    := E_CamAxisState.eCamAxisState_Error;
        ELSIF McCamIn.InSync THEN
            // InSync May Not Report Immediately Until Slave Axis Has Past Activation Point 

            //_StartSync := FALSE;
            McCamIn.Execute := FALSE;
            _RunningTable   := CurrentTableSelect;
            SequenceState   := E_CamAxisState.eCamAxisState_SetChangeMode;
        END_IF
    E_CamAxisState.eCamAxisState_SetChangeMode:
        MCSetCamOnlineChangeMode.Execute := TRUE;
        IF MCSetCamOnlineChangeMode.Error THEN
            //MCSetCamOnlineChangeMode.Execute := FALSE;
            SequenceErrorID := MCSetCamOnlineChangeMode.ErrorID;
            SequenceState   := E_CamAxisState.eCamAxisState_Error;
        ELSIF MCSetCamOnlineChangeMode.Done THEN
            MCSetCamOnlineChangeMode.Execute := FALSE;
            ChangeModeCommand                := FALSE;
            StartSyncCommand                 := FALSE;
            StartCoupleCommand               := FALSE;
            SequenceState                    := E_CamAxisState.eCamAxisState_WaitForChangeCommand;
        END_IF
    E_CamAxisState.eCamAxisState_WaitForChangeCommand:
        IF NOT _InSync THEN
            // Axis is No Longer Coupled 
            SequenceState := E_CamAxisState.eCamAxisState_WaitForCommand;
        ELSIF ChangeModeCommand THEN
            // Update OnLineChangeMode 
            SequenceState := E_CamAxisState.eCamAxisState_SetChangeMode;
        ELSIF _CamParameters.TableSelect <> OldTableSelect OR UpdateTableCommand THEN
            // Table Number Changed or Update Current Table 
            OldTableSelect := _CamParameters.TableSelect;
            IF _CamParameters.TableSelect < 1 OR _CamParameters.TableSelect > Parameters_MotionControl.CAM_SLAVE_AXIS_TABLES THEN
                SequenceState := E_CamAxisState.eCamAxisState_Error;
            ELSE
                // Update Points 
                CurrentTableSelect            := _CamParameters.TableSelect;
                CurrentPoints                 := _CamParameters.CamTable[CurrentTableSelect].Points;
                CurrentTable.pArray           := ADR(CurrentPoints);
                CurrentTable.ArraySize        := SIZEOF(CurrentPoints);
                CurrentTable.NoOfColumns      := 1;
                CurrentTable.NoOfRows         := DINT_TO_UDINT(_CamParameters.CamTable[CurrentTableSelect].NumberOfPoints);
                CurrentTable.TableType        := MC_TABLETYPE_MOTIONFUNCTION;
                McWriteMotionFunction.Execute := TRUE;
                UpdateTableCommand            := TRUE;
                SequenceState                 := E_CamAxisState.eCamAxisState_WriteNewTable;
            END_IF
        END_IF
    E_CamAxisState.eCamAxisState_WriteNewTable:
        IF NOT McWriteMotionFunction.Busy THEN
            McWriteMotionFunction.Execute := FALSE;
            IF McWriteMotionFunction.Error THEN
                SequenceErrorID := McWriteMotionFunction.ErrorID;
                SequenceState   := E_CamAxisState.eCamAxisState_Error;
            ELSIF McWriteMotionFunction.Done THEN
                SequenceState := E_CamAxisState.eCamAxisState_WaitForActive;
            END_IF
        END_IF
    E_CamAxisState.eCamAxisState_WaitForActive:
        IF NOT _Axis.Status.CamDataQueued OR NOT UpdateTableCommand THEN
            // Cam Data Queued Will Not Turn Off Until Master Has Gone Past The Activation Position 

            // Abort Waiting for New Table to Activate if _UpdateTable and _UpdateTableNow Are Both Off 
            UpdateTableCommand := FALSE;
            _RunningTable      := CurrentTableSelect;
            SequenceState      := E_CamAxisState.eCamAxisState_WaitForChangeCommand;
        END_IF
    E_CamAxisState.eCamAxisState_Error: // ERROR STATE 
        FindSlavePositionCommand := FALSE;
        FindSyncPositionCommand  := FALSE;
        StartSyncCommand         := FALSE;
        StartCoupleCommand       := FALSE;
        UpdateTableCommand       := FALSE;
        ChangeModeCommand        := FALSE;

        // Wait for Reset Input
        SequenceError := TRUE;
        _Error        := TRUE;
        _ErrorID      := SequenceErrorID;
END_CASE

//Call local FBs
SUPER^.CyclicLogic();
END_METHOD

METHOD PROTECTED CallFBs : BOOL
VAR_INPUT
END_VAR
SUPER^.CallFBs();
IF __ISVALIDREF(_CamParameters) AND __ISVALIDREF(_Master) THEN
    MCReadCamTableSlaveDynamics(CamTableID := _CamParameters.CamTableId, MasterPosition := ReadSlaveDynamicsMasterPos + _CamParameters.MasterOffset);
    MCCamTableSelect(Periodic       := _CamParameters.Periodic,
                     MasterAbsolute := TRUE, // Not Implemented 
                     SlaveAbsolute  := TRUE, // Not Implemented 
                     CamTableID     := _CamParameters.CamTableId,
                     Master         := _Master,
                     Slave          := _Axis,
                     CamTable       := CurrentTable);

    McWriteMotionFunction(CamTableID := _CamParameters.CamTableId,
                          PointID    := 1,
                          NumPoints  := DINT_TO_UDINT(_CamParameters.CamTable[CurrentTableSelect].NumberOfPoints),
                          CamTable   := CurrentTable);

    MCSetCamOnlineChangeMode(ActivationMode     := _CamParameters.ChangeOptions.ActivationMode,
                             ActivationPosition := _CamParameters.ChangeOptions.ActivationPosition,
                             MasterScalingMode  := _CamParameters.ChangeOptions.MasterScalingMode,
                             SlaveScalingMode   := _CamParameters.ChangeOptions.SlaveScalingMode,
                             CamTableID         := _CamParameters.CamTableId);

    McCamIn(MasterOffset  := _CamParameters.MasterOffset,
            SlaveOffset   := _CamParameters.SlaveOffset,
            MasterScaling := _CamParameters.MasterScaling,
            SlaveScaling  := _CamParameters.SlaveScaling,
            StartMode     := _CamParameters.StartMode,
            CamTableID    := _CamParameters.CamTableId,
            BufferMode    := _CamParameters.BufferMode,
            Options       := _CamParameters.CamInOptions,
            Master        := _Master,
            Slave         := _Axis);

    McCamOut(Slave := _Axis);
END_IF

// semaphore commands on while busy
SemaphoreBusy := StartSyncCommand OR StartCoupleCommand OR FindSlavePositionCommand OR FindSyncPositionCommand OR UpdateTableCommand OR ChangeModeCommand;

//SemaphoreBusy := StartSyncCommand OR StartCoupleCommand OR StopCommand OR FindSlavePositionCommand OR FindSyncPositionCommand OR UpdateTableCommand OR ChangeModeCommand;

// ceck for function blocks busy
_Busy := _Busy OR SemaphoreBusy OR MCReadParameterSet.Busy OR MCCamTableSelect.Busy OR McCamIn.Busy OR McCamOut.Busy OR MCReadCamTableSlaveDynamics.Busy OR MCSetCamOnlineChangeMode.Busy OR
         McWriteMotionFunction.Busy;
END_METHOD

METHOD PROTECTED Initialize : BOOL
VAR_INPUT
END_VAR
IF NOT __ISVALIDREF(_Master) THEN
    _Master REF= DummyAxis;
END_IF

Initialize := SUPER^.Initialize();
END_METHOD

END_FUNCTION_BLOCK

// Interfaces/I_CamSlaveAxis
INTERFACE I_CamSlaveAxis EXTENDS I_BasicAxis

PROPERTY CamParameters : REFERENCE TO ST_CamParameters
GET
END_GET
SET
END_SET
END_PROPERTY

METHOD ChangeMode : BOOL
VAR_INPUT
END_VAR
END_METHOD

METHOD FindSlavePos : BOOL
VAR_INPUT
END_VAR
END_METHOD

METHOD FindSyncPos : BOOL
VAR_INPUT
END_VAR
END_METHOD

PROPERTY InSync : BOOL
GET
END_GET
END_PROPERTY

PROPERTY Master : REFERENCE TO AXIS_REF
GET
END_GET
SET
END_SET
END_PROPERTY

PROPERTY RunningTable : UDINT
GET
END_GET
END_PROPERTY

METHOD StartCouple : BOOL
VAR_INPUT
END_VAR
END_METHOD

METHOD StartSync : BOOL
VAR_INPUT
END_VAR
END_METHOD

PROPERTY SyncPos : LREAL
GET
END_GET
END_PROPERTY

METHOD UpdateTable : BOOL
VAR_INPUT
END_VAR
END_METHOD

END_INTERFACE

// Project Information/F_GetCompany
// This function has been automatically generated from the project information.
{attribute 'signature_flag' := '1073741824'}
{attribute 'TcGenerated'}
{attribute 'no-analysis'}
FUNCTION F_GetCompany : WSTRING
VAR_INPUT
	
END_VAR

F_GetCompany := "Beckhoff Automation LLC";

END_FUNCTION

// Project Information/F_GetTitle
// This function has been automatically generated from the project information.
{attribute 'signature_flag' := '1073741824'}
{attribute 'TcGenerated'}
{attribute 'no-analysis'}
FUNCTION F_GetTitle : WSTRING
VAR_INPUT
	
END_VAR

F_GetTitle := "SPT Motion Control";

END_FUNCTION

// Project Information/F_GetVersion
// This function has been automatically generated from the project information.
{attribute 'signature_flag' := '1073741824'}
{attribute 'TcGenerated'}
{attribute 'no-analysis'}
FUNCTION F_GetVersion : ST_LibVersion
VAR_INPUT
	
END_VAR

F_GetVersion.iMajor := 3;
F_GetVersion.iMinor := 1;
F_GetVersion.iBuild := 0;
F_GetVersion.iRevision := 0;
F_GetVersion.sVersion := '3.1.0';
F_GetVersion.nFlags := 1;

END_FUNCTION
